LIN {X -0.164,Y -450.887,Z 1407.566,A 0.000,B 0.000,C 90.000,E1 281.951} C_DIS
LIN {X -0.109,Y -452.134,Z 1407.563,A 0.000,B 0.000,C 90.000,E1 281.422} C_DIS
LIN {X -0.046,Y -452.993,Z 1407.561,A 0.000,B 0.000,C 90.000,E1 280.894} C_DIS
LIN {X 0.023,Y -453.472,Z 1407.558,A 0.000,B 0.000,C 90.000,E1 280.366} C_DIS
LIN {X 0.016,Y -453.459,Z 1407.555,A 0.000,B 0.000,C 90.000,E1 279.849} C_DIS
LIN {X 0.091,Y -452.973,Z 1407.552,A 0.000,B 0.000,C 90.000,E1 279.321} C_DIS
LIN {X 0.091,Y -451.933,Z 1407.549,A 0.000,B 0.000,C 90.000,E1 278.803} C_DIS
LIN {X 0.156,Y -450.386,Z 1407.546,A 0.000,B 0.000,C 90.000,E1 278.276} C_DIS
LIN {X 0.149,Y -448.152,Z 1407.543,A 0.000,B 0.000,C 90.000,E1 277.757} C_DIS
LIN {X 0.128,Y -445.154,Z 1407.540,A 0.000,B 0.000,C 90.000,E1 277.239} C_DIS
LIN {X -0.082,Y -443.358,Z 1407.539,A 0.000,B 0.000,C 90.000,E1 277.004} C_DIS
LIN {X -0.126,Y -439.024,Z 1407.536,A 0.000,B 0.000,C 90.000,E1 276.486} C_DIS
LIN {X 0.042,Y -436.474,Z 1407.534,A 0.000,B 0.000,C 90.000,E1 276.201} C_DIS
LIN {X 0.046,Y -430.491,Z 1407.532,A 0.000,B 0.000,C 90.000,E1 275.682} C_DIS
LIN {X 0.146,Y -424.269,Z 1407.529,A 0.000,B 0.000,C 90.000,E1 275.220} C_DIS
LIN {X -0.212,Y -417.873,Z 1407.527,A 0.000,B 0.000,C 90.000,E1 274.878} C_DIS
LIN {X 0.190,Y -411.195,Z 1407.525,A 0.000,B 0.000,C 90.000,E1 274.473} C_DIS
LIN {X -0.124,Y -401.382,Z 1407.523,A 0.000,B 0.000,C 90.000,E1 274.073} C_DIS
LIN {X -0.064,Y -391.586,Z 1407.520,A 0.000,B 0.000,C 90.000,E1 273.669} C_DIS
LIN {X -0.077,Y -378.690,Z 1407.518,A 0.000,B 0.000,C 90.000,E1 273.212} C_DIS
LIN {X -0.178,Y -368.306,Z 1407.516,A 0.000,B 0.000,C 90.000,E1 272.922} C_DIS
LIN {X 0.035,Y -357.753,Z 1407.515,A 0.000,B 0.000,C 90.000,E1 272.636} C_DIS
LIN {X -0.170,Y -346.589,Z 1407.514,A 0.000,B 0.000,C 90.000,E1 272.465} C_DIS
LIN {X -0.105,Y -332.924,Z 1407.513,A 0.000,B 0.000,C 90.000,E1 272.293} C_DIS
LIN {X 0.118,Y -317.949,Z 1407.512,A 0.000,B 0.000,C 90.000,E1 272.178} C_DIS
LIN {X 0.057,Y -313.232,Z 1407.512,A 0.000,B 0.000,C 90.000,E1 272.178} C_DIS
LIN {X 0.014,Y -181.233,Z 1407.512,A 0.000,B 0.000,C 90.000,E1 272.178} C_DIS
LIN {X -0.010,Y -181.571,Z 1407.503,A 0.000,B 0.000,C 90.000,E1 270.458} C_DIS
LIN {X -0.090,Y -180.932,Z 1407.479,A 0.000,B 0.000,C 90.000,E1 266.274} C_DIS
LIN {X -0.032,Y -180.906,Z 1407.474,A 0.000,B 0.000,C 90.000,E1 265.412} C_DIS
LIN {X 0.041,Y -180.705,Z 1407.470,A 0.000,B 0.000,C 90.000,E1 264.546} C_DIS
LIN {X -0.056,Y -178.791,Z 1407.442,A 0.000,B 0.000,C 90.000,E1 259.511} C_DIS
LIN {X 0.020,Y -175.837,Z 1407.413,A 0.000,B 0.000,C 90.000,E1 254.393} C_DIS
LIN {X 0.021,Y -172.026,Z 1407.385,A 0.000,B 0.000,C 90.000,E1 249.263} C_DIS
LIN {X -0.003,Y -171.453,Z 1407.380,A 0.000,B 0.000,C 90.000,E1 248.411} C_DIS
LIN {X -0.023,Y -167.687,Z 1407.356,A 0.000,B 0.000,C 90.000,E1 244.101} C_DIS
LIN {X -0.009,Y -166.367,Z 1407.346,A 0.000,B 0.000,C 90.000,E1 242.359} C_DIS
LIN {X -0.017,Y -163.098,Z 1407.327,A 0.000,B 0.000,C 90.000,E1 238.869} C_DIS
LIN {X 0.034,Y -161.043,Z 1407.312,A 0.000,B 0.000,C 90.000,E1 236.215} C_DIS
LIN {X 0.018,Y -157.780,Z 1407.293,A 0.000,B 0.000,C 90.000,E1 232.683} C_DIS
LIN {X 0.080,Y -155.817,Z 1407.278,A 0.000,B 0.000,C 90.000,E1 229.989} C_DIS
LIN {X -0.081,Y -152.069,Z 1407.253,A 0.000,B 0.000,C 90.000,E1 225.567} C_DIS
LIN {X -0.062,Y -150.319,Z 1407.238,A 0.000,B 0.000,C 90.000,E1 222.852} C_DIS
LIN {X -0.040,Y -147.061,Z 1407.213,A 0.000,B 0.000,C 90.000,E1 218.302} C_DIS
LIN {X 0.067,Y -145.638,Z 1407.198,A 0.000,B 0.000,C 90.000,E1 215.518} C_DIS
LIN {X 0.065,Y -143.020,Z 1407.172,A 0.000,B 0.000,C 90.000,E1 210.924} C_DIS
LIN {X -0.004,Y -141.646,Z 1407.151,A 0.000,B 0.000,C 90.000,E1 207.257} C_DIS
LIN {X 0.046,Y -139.442,Z 1407.115,A 0.000,B 0.000,C 90.000,E1 200.737} C_DIS
LIN {X -0.032,Y -139.175,Z 1407.105,A 0.000,B 0.000,C 90.000,E1 198.906} C_DIS
LIN {X -0.004,Y -138.319,Z 1407.053,A 0.000,B 0.000,C 90.000,E1 189.557} C_DIS
LIN {X 0.006,Y -139.470,Z 1407.006,A 0.000,B 0.000,C 90.000,E1 181.146} C_DIS
LIN {X -0.054,Y -141.040,Z 1406.975,A 0.000,B 0.000,C 90.000,E1 175.584} C_DIS
LIN {X 0.041,Y -142.409,Z 1406.960,A 0.000,B 0.000,C 90.000,E1 172.761} C_DIS
LIN {X -0.038,Y -144.642,Z 1406.934,A 0.000,B 0.000,C 90.000,E1 168.173} C_DIS
LIN {X 0.022,Y -147.839,Z 1406.909,A 0.000,B 0.000,C 90.000,E1 163.559} C_DIS
LIN {X -0.034,Y -150.536,Z 1406.888,A 0.000,B 0.000,C 90.000,E1 159.934} C_DIS
LIN {X -0.016,Y -154.000,Z 1406.868,A 0.000,B 0.000,C 90.000,E1 156.305} C_DIS
LIN {X 0.045,Y -157.413,Z 1406.848,A 0.000,B 0.000,C 90.000,E1 152.692} C_DIS
LIN {X 0.067,Y -161.624,Z 1406.829,A 0.000,B 0.000,C 90.000,E1 149.125} C_DIS
LIN {X 0.086,Y -165.819,Z 1406.809,A 0.000,B 0.000,C 90.000,E1 145.595} C_DIS
LIN {X 0.079,Y -170.788,Z 1406.790,A 0.000,B 0.000,C 90.000,E1 142.110} C_DIS
LIN {X -0.004,Y -175.659,Z 1406.771,A 0.000,B 0.000,C 90.000,E1 138.690} C_DIS
LIN {X -0.007,Y -181.273,Z 1406.752,A 0.000,B 0.000,C 90.000,E1 135.283} C_DIS
LIN {X -0.007,Y -186.748,Z 1406.733,A 0.000,B 0.000,C 90.000,E1 131.919} C_DIS
LIN {X -0.056,Y -191.344,Z 1406.719,A 0.000,B 0.000,C 90.000,E1 129.439} C_DIS
LIN {X -0.010,Y -197.180,Z 1406.701,A 0.000,B 0.000,C 90.000,E1 126.137} C_DIS
LIN {X 0.015,Y -199.638,Z 1406.694,A 0.000,B 0.000,C 90.000,E1 124.898} C_DIS
LIN {X -0.011,Y -310.460,Z 1406.694,A 0.000,B 0.000,C 90.000,E1 124.898} C_DIS
LIN {X 0.052,Y -316.081,Z 1406.693,A 0.000,B 0.000,C 90.000,E1 124.692} C_DIS
LIN {X 0.117,Y -318.647,Z 1406.692,A 0.000,B 0.000,C 90.000,E1 124.485} C_DIS
LIN {X -0.078,Y -322.451,Z 1406.689,A 0.000,B 0.000,C 90.000,E1 124.072} C_DIS
LIN {X 0.211,Y -324.301,Z 1406.688,A 0.000,B 0.000,C 90.000,E1 123.706} C_DIS
LIN {X 0.047,Y -325.742,Z 1406.686,A 0.000,B 0.000,C 90.000,E1 123.420} C_DIS
LIN {X -0.157,Y -338.662,Z 1406.667,A 0.000,B 0.000,C 90.000,E1 120.001} C_DIS
LIN {X -0.002,Y -350.683,Z 1406.651,A 0.000,B 0.000,C 90.000,E1 117.206} C_DIS
LIN {X -0.134,Y -364.162,Z 1406.636,A 0.000,B 0.000,C 90.000,E1 114.515} C_DIS
LIN {X -0.121,Y -377.467,Z 1406.623,A 0.000,B 0.000,C 90.000,E1 112.153} C_DIS
LIN {X 0.091,Y -392.109,Z 1406.610,A 0.000,B 0.000,C 90.000,E1 109.812} C_DIS
LIN {X -0.098,Y -408.194,Z 1406.598,A 0.000,B 0.000,C 90.000,E1 107.583} C_DIS
LIN {X -0.012,Y -425.832,Z 1406.585,A 0.000,B 0.000,C 90.000,E1 105.371} C_DIS
LIN {X -0.082,Y -445.088,Z 1406.573,A 0.000,B 0.000,C 90.000,E1 103.244} C_DIS
LIN {X 0.011,Y -465.219,Z 1406.563,A 0.000,B 0.000,C 90.000,E1 101.243} C_DIS
LIN {X 0.182,Y -483.286,Z 1406.553,A 0.000,B 0.000,C 90.000,E1 99.613} C_DIS
LIN {X -0.157,Y -485.624,Z 1406.552,A 0.000,B 0.000,C 90.000,E1 99.434} C_DIS
LIN {X -0.097,Y -487.395,Z 1406.551,A 0.000,B 0.000,C 90.000,E1 99.208} C_DIS
LIN {X -0.205,Y -488.920,Z 1406.550,A 0.000,B 0.000,C 90.000,E1 98.973} C_DIS
LIN {X 0.096,Y -490.057,Z 1406.548,A 0.000,B 0.000,C 90.000,E1 98.690} C_DIS
LIN {X -0.102,Y -491.406,Z 1406.546,A 0.000,B 0.000,C 90.000,E1 98.219} C_DIS
LIN {X 0.121,Y -491.715,Z 1406.543,A 0.000,B 0.000,C 90.000,E1 97.701} C_DIS
LIN {X -0.136,Y -491.034,Z 1406.540,A 0.000,B 0.000,C 90.000,E1 97.239} C_DIS
LIN {X 0.097,Y -489.256,Z 1406.537,A 0.000,B 0.000,C 90.000,E1 96.720} C_DIS
LIN {X -0.004,Y -487.849,Z 1406.536,A 0.000,B 0.000,C 90.000,E1 96.486} C_DIS
LIN {X -0.036,Y -468.285,Z 1406.519,A 0.000,B 0.000,C 90.000,E1 93.498} C_DIS
LIN {X 0.108,Y -461.753,Z 1406.514,A 0.000,B 0.000,C 90.000,E1 92.465} C_DIS
LIN {X -0.208,Y -440.357,Z 1406.495,A 0.000,B 0.000,C 90.000,E1 89.141} C_DIS
LIN {X 0.076,Y -429.683,Z 1406.485,A 0.000,B 0.000,C 90.000,E1 87.249} C_DIS
LIN {X 0.154,Y -418.808,Z 1406.474,A 0.000,B 0.000,C 90.000,E1 85.355} C_DIS
LIN {X 0.081,Y -407.789,Z 1406.464,A 0.000,B 0.000,C 90.000,E1 83.451} C_DIS
LIN {X 0.192,Y -396.699,Z 1406.453,A 0.000,B 0.000,C 90.000,E1 81.489} C_DIS
LIN {X 0.132,Y -387.026,Z 1406.443,A 0.000,B 0.000,C 90.000,E1 79.803} C_DIS
LIN {X -0.003,Y -375.657,Z 1406.432,A 0.000,B 0.000,C 90.000,E1 77.813} C_DIS
LIN {X 0.077,Y -364.284,Z 1406.421,A 0.000,B 0.000,C 90.000,E1 75.755} C_DIS
LIN {X 0.049,Y -354.447,Z 1406.411,A 0.000,B 0.000,C 90.000,E1 73.976} C_DIS
LIN {X -0.058,Y -344.544,Z 1406.401,A 0.000,B 0.000,C 90.000,E1 72.181} C_DIS
LIN {X 0.078,Y -334.556,Z 1406.391,A 0.000,B 0.000,C 90.000,E1 70.315} C_DIS
LIN {X 0.057,Y -318.235,Z 1406.373,A 0.000,B 0.000,C 90.000,E1 67.177} C_DIS
LIN {X 0.021,Y -304.503,Z 1406.357,A 0.000,B 0.000,C 90.000,E1 64.280} C_DIS
LIN {X 0.023,Y -293.573,Z 1406.343,A 0.000,B 0.000,C 90.000,E1 61.641} C_DIS
LIN {X -0.024,Y -281.325,Z 1406.324,A 0.000,B 0.000,C 90.000,E1 58.280} C_DIS
LIN {X -0.014,Y -271.322,Z 1406.307,A 0.000,B 0.000,C 90.000,E1 55.182} C_DIS
LIN {X -0.104,Y -260.957,Z 1406.287,A 0.000,B 0.000,C 90.000,E1 51.698} C_DIS
LIN {X 0.091,Y -251.179,Z 1406.267,A 0.000,B 0.000,C 90.000,E1 48.081} C_DIS
LIN {X 0.115,Y -242.158,Z 1406.247,A 0.000,B 0.000,C 90.000,E1 44.433} C_DIS
LIN {X 0.036,Y -234.059,Z 1406.226,A 0.000,B 0.000,C 90.000,E1 40.744} C_DIS
LIN {X -0.040,Y -226.822,Z 1406.205,A 0.000,B 0.000,C 90.000,E1 36.996} C_DIS
LIN {X -0.010,Y -220.392,Z 1406.184,A 0.000,B 0.000,C 90.000,E1 33.166} C_DIS
LIN {X 0.026,Y -214.864,Z 1406.163,A 0.000,B 0.000,C 90.000,E1 29.283} C_DIS
LIN {X 0.135,Y -210.199,Z 1406.141,A 0.000,B 0.000,C 90.000,E1 25.335} C_DIS
LIN {X 0.044,Y -205.914,Z 1406.115,A 0.000,B 0.000,C 90.000,E1 20.610} C_DIS
LIN {X -0.045,Y -202.753,Z 1406.088,A 0.000,B 0.000,C 90.000,E1 15.843} C_DIS
LIN {X -0.046,Y -200.755,Z 1406.066,A 0.000,B 0.000,C 90.000,E1 11.827} C_DIS
LIN {X 0.077,Y -199.136,Z 1406.043,A 0.000,B 0.000,C 90.000,E1 7.757} C_DIS
LIN {X 0.020,Y -197.815,Z 1406.021,A 0.000,B 0.000,C 90.000,E1 3.726} C_DIS
LIN {X -0.036,Y -196.886,Z 1405.997,A 0.000,B 0.000,C 90.000,E1 359.542} C_DIS
LIN {X -0.050,Y -196.289,Z 1405.970,A 0.000,B 0.000,C 90.000,E1 354.666} C_DIS
LIN {X 0.067,Y -196.501,Z 1405.943,A 0.000,B 0.000,C 90.000,E1 349.746} C_DIS
LIN {X 0.116,Y -198.640,Z 1405.902,A 0.000,B 0.000,C 90.000,E1 342.417} C_DIS
LIN {X -0.055,Y -201.702,Z 1405.875,A 0.000,B 0.000,C 90.000,E1 337.614} C_DIS
LIN {X -0.023,Y -205.507,Z 1405.853,A 0.000,B 0.000,C 90.000,E1 333.589} C_DIS
LIN {X -0.055,Y -210.394,Z 1405.831,A 0.000,B 0.000,C 90.000,E1 329.616} C_DIS
LIN {X -0.040,Y -216.574,Z 1405.809,A 0.000,B 0.000,C 90.000,E1 325.674} C_DIS
LIN {X -0.019,Y -222.598,Z 1405.792,A 0.000,B 0.000,C 90.000,E1 322.557} C_DIS
LIN {X 0.080,Y -229.516,Z 1405.775,A 0.000,B 0.000,C 90.000,E1 319.461} C_DIS
LIN {X 0.117,Y -238.333,Z 1405.756,A 0.000,B 0.000,C 90.000,E1 316.053} C_DIS
LIN {X -0.096,Y -248.303,Z 1405.738,A 0.000,B 0.000,C 90.000,E1 312.771} C_DIS
LIN {X -0.027,Y -258.345,Z 1405.721,A 0.000,B 0.000,C 90.000,E1 309.850} C_DIS
LIN {X -0.088,Y -270.900,Z 1405.704,A 0.000,B 0.000,C 90.000,E1 306.664} C_DIS
LIN {X 0.116,Y -280.302,Z 1405.692,A 0.000,B 0.000,C 90.000,E1 304.532} C_DIS
LIN {X 0.091,Y -287.165,Z 1405.684,A 0.000,B 0.000,C 90.000,E1 303.166} C_DIS
LIN {X 0.144,Y -296.748,Z 1405.675,A 0.000,B 0.000,C 90.000,E1 301.465} C_DIS
LIN {X 0.175,Y -305.354,Z 1405.668,A 0.000,B 0.000,C 90.000,E1 300.129} C_DIS
LIN {X -0.112,Y -314.850,Z 1405.660,A 0.000,B 0.000,C 90.000,E1 298.871} C_DIS
LIN {X -0.129,Y -325.425,Z 1405.653,A 0.000,B 0.000,C 90.000,E1 297.590} C_DIS
LIN {X -0.149,Y -347.264,Z 1405.640,A 0.000,B 0.000,C 90.000,E1 295.207} C_DIS
LIN {X -0.068,Y -360.771,Z 1405.632,A 0.000,B 0.000,C 90.000,E1 293.770} C_DIS
LIN {X -0.063,Y -371.276,Z 1405.626,A 0.000,B 0.000,C 90.000,E1 292.642} C_DIS
LIN {X 0.059,Y -381.612,Z 1405.619,A 0.000,B 0.000,C 90.000,E1 291.482} C_DIS
LIN {X -0.077,Y -394.201,Z 1405.611,A 0.000,B 0.000,C 90.000,E1 290.066} C_DIS
LIN {X 0.079,Y -414.125,Z 1405.599,A 0.000,B 0.000,C 90.000,E1 287.819} C_DIS
LIN {X 0.165,Y -421.495,Z 1405.594,A 0.000,B 0.000,C 90.000,E1 286.985} C_DIS
LIN {X -0.032,Y -428.273,Z 1405.590,A 0.000,B 0.000,C 90.000,E1 286.205} C_DIS
LIN {X -0.001,Y -432.410,Z 1405.587,A 0.000,B 0.000,C 90.000,E1 285.662} C_DIS
LIN {X -0.063,Y -436.154,Z 1405.584,A 0.000,B 0.000,C 90.000,E1 285.134} C_DIS
LIN {X 0.219,Y -441.051,Z 1405.580,A 0.000,B 0.000,C 90.000,E1 284.300} C_DIS
LIN {X -0.215,Y -443.860,Z 1405.577,A 0.000,B 0.000,C 90.000,E1 283.828} C_DIS
LIN {X 0.027,Y -447.401,Z 1405.572,A 0.000,B 0.000,C 90.000,E1 283.008} C_DIS
LIN {X 0.067,Y -449.377,Z 1405.569,A 0.000,B 0.000,C 90.000,E1 282.479} C_DIS
LIN {X 0.112,Y -450.991,Z 1405.567,A 0.000,B 0.000,C 90.000,E1 281.951} C_DIS
LIN {X 0.169,Y -452.230,Z 1405.564,A 0.000,B 0.000,C 90.000,E1 281.422} C_DIS
LIN {X -0.212,Y -453.131,Z 1405.561,A 0.000,B 0.000,C 90.000,E1 280.950} C_DIS
LIN {X -0.142,Y -453.645,Z 1405.558,A 0.000,B 0.000,C 90.000,E1 280.423} C_DIS
LIN {X -0.150,Y -453.657,Z 1405.555,A 0.000,B 0.000,C 90.000,E1 279.905} C_DIS
LIN {X -0.075,Y -453.234,Z 1405.552,A 0.000,B 0.000,C 90.000,E1 279.378} C_DIS
LIN {X -0.074,Y -452.292,Z 1405.549,A 0.000,B 0.000,C 90.000,E1 278.859} C_DIS
LIN {X -0.071,Y -450.785,Z 1405.546,A 0.000,B 0.000,C 90.000,E1 278.341} C_DIS
LIN {X -0.012,Y -448.649,Z 1405.543,A 0.000,B 0.000,C 90.000,E1 277.814} C_DIS
LIN {X -0.024,Y -445.765,Z 1405.541,A 0.000,B 0.000,C 90.000,E1 277.296} C_DIS
LIN {X -0.054,Y -442.041,Z 1405.538,A 0.000,B 0.000,C 90.000,E1 276.777} C_DIS
LIN {X -0.102,Y -437.324,Z 1405.535,A 0.000,B 0.000,C 90.000,E1 276.258} C_DIS
LIN {X 0.115,Y -434.562,Z 1405.533,A 0.000,B 0.000,C 90.000,E1 275.967} C_DIS
LIN {X -0.139,Y -428.517,Z 1405.531,A 0.000,B 0.000,C 90.000,E1 275.511} C_DIS
LIN {X 0.120,Y -422.247,Z 1405.528,A 0.000,B 0.000,C 90.000,E1 275.049} C_DIS
LIN {X -0.075,Y -415.762,Z 1405.526,A 0.000,B 0.000,C 90.000,E1 274.702} C_DIS
LIN {X 0.148,Y -405.811,Z 1405.523,A 0.000,B 0.000,C 90.000,E1 274.188} C_DIS
LIN {X 0.094,Y -396.109,Z 1405.521,A 0.000,B 0.000,C 90.000,E1 273.784} C_DIS
LIN {X -0.108,Y -386.263,Z 1405.519,A 0.000,B 0.000,C 90.000,E1 273.440} C_DIS
LIN {X -0.010,Y -376.360,Z 1405.517,A 0.000,B 0.000,C 90.000,E1 273.094} C_DIS
LIN {X 0.172,Y -369.429,Z 1405.516,A 0.000,B 0.000,C 90.000,E1 272.865} C_DIS
LIN {X 0.019,Y -358.758,Z 1405.515,A 0.000,B 0.000,C 90.000,E1 272.636} C_DIS
LIN {X 0.165,Y -347.772,Z 1405.514,A 0.000,B 0.000,C 90.000,E1 272.407} C_DIS
LIN {X -0.119,Y -334.120,Z 1405.513,A 0.000,B 0.000,C 90.000,E1 272.293} C_DIS
LIN {X 0.108,Y -321.060,Z 1405.512,A 0.000,B 0.000,C 90.000,E1 272.178} C_DIS
LIN {X 0.010,Y -313.166,Z 1405.512,A 0.000,B 0.000,C 90.000,E1 272.178} C_DIS
LIN {X -0.016,Y -181.234,Z 1405.512,A 0.000,B 0.000,C 90.000,E1 272.178} C_DIS
LIN {X -0.034,Y -181.572,Z 1405.502,A 0.000,B 0.000,C 90.000,E1 270.458} C_DIS
LIN {X -0.056,Y -180.906,Z 1405.474,A 0.000,B 0.000,C 90.000,E1 265.412} C_DIS
LIN {X 0.018,Y -180.701,Z 1405.470,A 0.000,B 0.000,C 90.000,E1 264.546} C_DIS
LIN {X -0.081,Y -178.786,Z 1405.442,A 0.000,B 0.000,C 90.000,E1 259.511} C_DIS
LIN {X -0.003,Y -175.833,Z 1405.413,A 0.000,B 0.000,C 90.000,E1 254.393} C_DIS
LIN {X -0.002,Y -172.022,Z 1405.385,A 0.000,B 0.000,C 90.000,E1 249.263} C_DIS
LIN {X -0.026,Y -171.447,Z 1405.380,A 0.000,B 0.000,C 90.000,E1 248.411} C_DIS
LIN {X 0.028,Y -167.681,Z 1405.356,A 0.000,B 0.000,C 90.000,E1 244.076} C_DIS
LIN {X -0.032,Y -166.358,Z 1405.346,A 0.000,B 0.000,C 90.000,E1 242.359} C_DIS
LIN {X -0.039,Y -163.091,Z 1405.327,A 0.000,B 0.000,C 90.000,E1 238.869} C_DIS
LIN {X 0.012,Y -161.035,Z 1405.312,A 0.000,B 0.000,C 90.000,E1 236.215} C_DIS
LIN {X -0.005,Y -157.774,Z 1405.293,A 0.000,B 0.000,C 90.000,E1 232.683} C_DIS
LIN {X 0.058,Y -155.812,Z 1405.278,A 0.000,B 0.000,C 90.000,E1 229.989} C_DIS
LIN {X 0.006,Y -152.063,Z 1405.253,A 0.000,B 0.000,C 90.000,E1 225.526} C_DIS
LIN {X -0.083,Y -150.313,Z 1405.238,A 0.000,B 0.000,C 90.000,E1 222.852} C_DIS
LIN {X 0.054,Y -147.056,Z 1405.213,A 0.000,B 0.000,C 90.000,E1 218.257} C_DIS
LIN {X 0.046,Y -145.634,Z 1405.197,A 0.000,B 0.000,C 90.000,E1 215.518} C_DIS
LIN {X 0.045,Y -143.017,Z 1405.172,A 0.000,B 0.000,C 90.000,E1 210.924} C_DIS
LIN {X -0.025,Y -141.643,Z 1405.151,A 0.000,B 0.000,C 90.000,E1 207.257} C_DIS
LIN {X 0.026,Y -139.440,Z 1405.115,A 0.000,B 0.000,C 90.000,E1 200.737} C_DIS
LIN {X -0.052,Y -139.173,Z 1405.105,A 0.000,B 0.000,C 90.000,E1 198.906} C_DIS
LIN {X -0.024,Y -138.318,Z 1405.053,A 0.000,B 0.000,C 90.000,E1 189.557} C_DIS
LIN {X -0.015,Y -139.472,Z 1405.006,A 0.000,B 0.000,C 90.000,E1 181.146} C_DIS
LIN {X 0.066,Y -141.044,Z 1404.975,A 0.000,B 0.000,C 90.000,E1 175.527} C_DIS
LIN {X 0.021,Y -142.413,Z 1404.960,A 0.000,B 0.000,C 90.000,E1 172.761} C_DIS
LIN {X -0.059,Y -144.648,Z 1404.934,A 0.000,B 0.000,C 90.000,E1 168.173} C_DIS
LIN {X 0.001,Y -147.844,Z 1404.909,A 0.000,B 0.000,C 90.000,E1 163.559} C_DIS
LIN {X -0.056,Y -150.543,Z 1404.888,A 0.000,B 0.000,C 90.000,E1 159.934} C_DIS
LIN {X -0.037,Y -154.008,Z 1404.868,A 0.000,B 0.000,C 90.000,E1 156.305} C_DIS
LIN {X 0.022,Y -157.423,Z 1404.848,A 0.000,B 0.000,C 90.000,E1 152.692} C_DIS
LIN {X 0.045,Y -161.634,Z 1404.829,A 0.000,B 0.000,C 90.000,E1 149.125} C_DIS
LIN {X 0.063,Y -165.829,Z 1404.809,A 0.000,B 0.000,C 90.000,E1 145.595} C_DIS
LIN {X 0.055,Y -170.800,Z 1404.790,A 0.000,B 0.000,C 90.000,E1 142.110} C_DIS
LIN {X -0.027,Y -175.670,Z 1404.771,A 0.000,B 0.000,C 90.000,E1 138.690} C_DIS
LIN {X 0.097,Y -181.284,Z 1404.751,A 0.000,B 0.000,C 90.000,E1 135.243} C_DIS
LIN {X -0.031,Y -186.762,Z 1404.733,A 0.000,B 0.000,C 90.000,E1 131.919} C_DIS
LIN {X 0.041,Y -191.356,Z 1404.719,A 0.000,B 0.000,C 90.000,E1 129.402} C_DIS
LIN {X -0.035,Y -197.194,Z 1404.701,A 0.000,B 0.000,C 90.000,E1 126.137} C_DIS
LIN {X 0.077,Y -199.601,Z 1404.694,A 0.000,B 0.000,C 90.000,E1 124.898} C_DIS
LIN {X 0.087,Y -310.119,Z 1404.694,A 0.000,B 0.000,C 90.000,E1 124.898} C_DIS
LIN {X -0.048,Y -311.871,Z 1404.694,A 0.000,B 0.000,C 90.000,E1 124.898} C_DIS
LIN {X 0.013,Y -316.366,Z 1404.693,A 0.000,B 0.000,C 90.000,E1 124.692} C_DIS
LIN {X 0.077,Y -318.822,Z 1404.692,A 0.000,B 0.000,C 90.000,E1 124.485} C_DIS
LIN {X -0.034,Y -322.641,Z 1404.689,A 0.000,B 0.000,C 90.000,E1 124.040} C_DIS
LIN {X 0.042,Y -324.457,Z 1404.687,A 0.000,B 0.000,C 90.000,E1 123.706} C_DIS
LIN {X 0.121,Y -325.868,Z 1404.686,A 0.000,B 0.000,C 90.000,E1 123.372} C_DIS
LIN {X -0.035,Y -337.529,Z 1404.668,A 0.000,B 0.000,C 90.000,E1 120.256} C_DIS
LIN {X 0.090,Y -349.408,Z 1404.653,A 0.000,B 0.000,C 90.000,E1 117.462} C_DIS
LIN {X -0.078,Y -362.742,Z 1404.638,A 0.000,B 0.000,C 90.000,E1 114.771} C_DIS
LIN {X 0.047,Y -375.903,Z 1404.624,A 0.000,B 0.000,C 90.000,E1 112.386} C_DIS
LIN {X 0.083,Y -390.393,Z 1404.612,A 0.000,B 0.000,C 90.000,E1 110.066} C_DIS
LIN {X -0.017,Y -406.312,Z 1404.599,A 0.000,B 0.000,C 90.000,E1 107.819} C_DIS
LIN {X 0.023,Y -423.773,Z 1404.587,A 0.000,B 0.000,C 90.000,E1 105.607} C_DIS
LIN {X -0.026,Y -442.876,Z 1404.575,A 0.000,B 0.000,C 90.000,E1 103.467} C_DIS
LIN {X -0.190,Y -462.943,Z 1404.564,A 0.000,B 0.000,C 90.000,E1 101.478} C_DIS
LIN {X -0.029,Y -483.550,Z 1404.553,A 0.000,B 0.000,C 90.000,E1 99.613} C_DIS
LIN {X 0.112,Y -485.789,Z 1404.552,A 0.000,B 0.000,C 90.000,E1 99.378} C_DIS
LIN {X 0.175,Y -487.486,Z 1404.551,A 0.000,B 0.000,C 90.000,E1 99.151} C_DIS
LIN {X 0.069,Y -488.951,Z 1404.550,A 0.000,B 0.000,C 90.000,E1 98.916} C_DIS
LIN {X -0.038,Y -490.040,Z 1404.548,A 0.000,B 0.000,C 90.000,E1 98.681} C_DIS
LIN {X 0.176,Y -491.312,Z 1404.545,A 0.000,B 0.000,C 90.000,E1 98.163} C_DIS
LIN {X -0.090,Y -491.553,Z 1404.543,A 0.000,B 0.000,C 90.000,E1 97.701} C_DIS
LIN {X 0.141,Y -490.804,Z 1404.540,A 0.000,B 0.000,C 90.000,E1 97.182} C_DIS
LIN {X -0.113,Y -488.940,Z 1404.537,A 0.000,B 0.000,C 90.000,E1 96.720} C_DIS
LIN {X -0.214,Y -487.476,Z 1404.536,A 0.000,B 0.000,C 90.000,E1 96.486} C_DIS
LIN {X 0.217,Y -467.918,Z 1404.519,A 0.000,B 0.000,C 90.000,E1 93.440} C_DIS
LIN {X 0.145,Y -459.666,Z 1404.512,A 0.000,B 0.000,C 90.000,E1 92.178} C_DIS
LIN {X 0.012,Y -439.998,Z 1404.495,A 0.000,B 0.000,C 90.000,E1 89.083} C_DIS
LIN {X -0.146,Y -429.339,Z 1404.485,A 0.000,B 0.000,C 90.000,E1 87.249} C_DIS
LIN {X -0.068,Y -418.503,Z 1404.474,A 0.000,B 0.000,C 90.000,E1 85.355} C_DIS
LIN {X -0.142,Y -407.532,Z 1404.464,A 0.000,B 0.000,C 90.000,E1 83.451} C_DIS
LIN {X -0.030,Y -396.456,Z 1404.453,A 0.000,B 0.000,C 90.000,E1 81.489} C_DIS
LIN {X -0.088,Y -386.792,Z 1404.443,A 0.000,B 0.000,C 90.000,E1 79.803} C_DIS
LIN {X 0.145,Y -375.453,Z 1404.432,A 0.000,B 0.000,C 90.000,E1 77.757} C_DIS
LIN {X -0.139,Y -364.079,Z 1404.421,A 0.000,B 0.000,C 90.000,E1 75.755} C_DIS
LIN {X -0.165,Y -354.215,Z 1404.411,A 0.000,B 0.000,C 90.000,E1 73.976} C_DIS
LIN {X 0.057,Y -344.308,Z 1404.401,A 0.000,B 0.000,C 90.000,E1 72.127} C_DIS
LIN {X -0.019,Y -334.294,Z 1404.391,A 0.000,B 0.000,C 90.000,E1 70.296} C_DIS
LIN {X -0.151,Y -317.969,Z 1404.373,A 0.000,B 0.000,C 90.000,E1 67.177} C_DIS
LIN {X 0.121,Y -302.841,Z 1404.355,A 0.000,B 0.000,C 90.000,E1 63.896} C_DIS
LIN {X 0.080,Y -292.078,Z 1404.340,A 0.000,B 0.000,C 90.000,E1 61.257} C_DIS
LIN {X 0.126,Y -280.013,Z 1404.322,A 0.000,B 0.000,C 90.000,E1 57.867} C_DIS
LIN {X 0.011,Y -271.202,Z 1404.306,A 0.000,B 0.000,C 90.000,E1 55.135} C_DIS
LIN {X 0.069,Y -260.886,Z 1404.287,A 0.000,B 0.000,C 90.000,E1 51.618} C_DIS
LIN {X -0.097,Y -251.135,Z 1404.267,A 0.000,B 0.000,C 90.000,E1 48.081} C_DIS
LIN {X -0.068,Y -242.146,Z 1404.247,A 0.000,B 0.000,C 90.000,E1 44.433} C_DIS
LIN {X 0.037,Y -234.077,Z 1404.226,A 0.000,B 0.000,C 90.000,E1 40.701} C_DIS
LIN {X -0.030,Y -226.866,Z 1404.205,A 0.000,B 0.000,C 90.000,E1 36.950} C_DIS
LIN {X 0.131,Y -220.480,Z 1404.184,A 0.000,B 0.000,C 90.000,E1 33.086} C_DIS
LIN {X -0.026,Y -214.981,Z 1404.162,A 0.000,B 0.000,C 90.000,E1 29.255} C_DIS
LIN {X -0.015,Y -210.377,Z 1404.141,A 0.000,B 0.000,C 90.000,E1 25.335} C_DIS
LIN {X -0.096,Y -206.140,Z 1404.114,A 0.000,B 0.000,C 90.000,E1 20.610} C_DIS
LIN {X 0.022,Y -203.037,Z 1404.088,A 0.000,B 0.000,C 90.000,E1 15.788} C_DIS
LIN {X 0.032,Y -201.072,Z 1404.065,A 0.000,B 0.000,C 90.000,E1 11.771} C_DIS
LIN {X -0.030,Y -199.452,Z 1404.043,A 0.000,B 0.000,C 90.000,E1 7.757} C_DIS
LIN {X -0.078,Y -198.140,Z 1404.021,A 0.000,B 0.000,C 90.000,E1 3.726} C_DIS
LIN {X -0.036,Y -197.190,Z 1403.997,A 0.000,B 0.000,C 90.000,E1 359.542} C_DIS
LIN {X -0.040,Y -196.550,Z 1403.970,A 0.000,B 0.000,C 90.000,E1 354.666} C_DIS
LIN {X 0.087,Y -196.734,Z 1403.943,A 0.000,B 0.000,C 90.000,E1 349.746} C_DIS
LIN {X -0.100,Y -198.883,Z 1403.903,A 0.000,B 0.000,C 90.000,E1 342.489} C_DIS
LIN {X -0.012,Y -201.927,Z 1403.876,A 0.000,B 0.000,C 90.000,E1 337.614} C_DIS
LIN {X 0.027,Y -205.729,Z 1403.853,A 0.000,B 0.000,C 90.000,E1 333.589} C_DIS
LIN {X 0.005,Y -210.613,Z 1403.831,A 0.000,B 0.000,C 90.000,E1 329.616} C_DIS
LIN {X 0.028,Y -216.789,Z 1403.809,A 0.000,B 0.000,C 90.000,E1 325.674} C_DIS
LIN {X 0.035,Y -221.194,Z 1403.796,A 0.000,B 0.000,C 90.000,E1 323.336} C_DIS
LIN {X -0.040,Y -227.890,Z 1403.779,A 0.000,B 0.000,C 90.000,E1 320.275} C_DIS
LIN {X -0.047,Y -236.448,Z 1403.760,A 0.000,B 0.000,C 90.000,E1 316.863} C_DIS
LIN {X 0.021,Y -246.105,Z 1403.742,A 0.000,B 0.000,C 90.000,E1 313.500} C_DIS
LIN {X -0.150,Y -255.833,Z 1403.725,A 0.000,B 0.000,C 90.000,E1 310.620} C_DIS
LIN {X 0.045,Y -268.089,Z 1403.708,A 0.000,B 0.000,C 90.000,E1 307.363} C_DIS
LIN {X 0.034,Y -277.137,Z 1403.696,A 0.000,B 0.000,C 90.000,E1 305.264} C_DIS
LIN {X -0.153,Y -285.453,Z 1403.686,A 0.000,B 0.000,C 90.000,E1 303.579} C_DIS
LIN {X -0.129,Y -294.774,Z 1403.677,A 0.000,B 0.000,C 90.000,E1 301.878} C_DIS
LIN {X -0.130,Y -303.168,Z 1403.670,A 0.000,B 0.000,C 90.000,E1 300.541} C_DIS
LIN {X -0.022,Y -312.381,Z 1403.662,A 0.000,B 0.000,C 90.000,E1 299.205} C_DIS
LIN {X -0.059,Y -319.685,Z 1403.657,A 0.000,B 0.000,C 90.000,E1 298.281} C_DIS
LIN {X 0.030,Y -344.032,Z 1403.642,A 0.000,B 0.000,C 90.000,E1 295.540} C_DIS
LIN {X -0.110,Y -357.565,Z 1403.634,A 0.000,B 0.000,C 90.000,E1 294.131} C_DIS
LIN {X -0.102,Y -368.124,Z 1403.628,A 0.000,B 0.000,C 90.000,E1 293.003} C_DIS
LIN {X 0.031,Y -378.528,Z 1403.621,A 0.000,B 0.000,C 90.000,E1 291.844} C_DIS
LIN {X -0.088,Y -391.142,Z 1403.613,A 0.000,B 0.000,C 90.000,E1 290.429} C_DIS
LIN {X 0.203,Y -408.577,Z 1403.602,A 0.000,B 0.000,C 90.000,E1 288.417} C_DIS
LIN {X -0.207,Y -418.361,Z 1403.597,A 0.000,B 0.000,C 90.000,E1 287.402} C_DIS
LIN {X 0.028,Y -425.472,Z 1403.592,A 0.000,B 0.000,C 90.000,E1 286.551} C_DIS
LIN {X 0.082,Y -431.912,Z 1403.588,A 0.000,B 0.000,C 90.000,E1 285.733} C_DIS
LIN {X -0.095,Y -437.493,Z 1403.583,A 0.000,B 0.000,C 90.000,E1 284.954} C_DIS
LIN {X 0.192,Y -442.247,Z 1403.579,A 0.000,B 0.000,C 90.000,E1 284.120} C_DIS
LIN {X -0.010,Y -446.124,Z 1403.574,A 0.000,B 0.000,C 90.000,E1 283.355} C_DIS
LIN {X -0.183,Y -449.278,Z 1403.570,A 0.000,B 0.000,C 90.000,E1 282.591} C_DIS
LIN {X -0.141,Y -450.930,Z 1403.567,A 0.000,B 0.000,C 90.000,E1 282.063} C_DIS
LIN {X -0.087,Y -452.258,Z 1403.564,A 0.000,B 0.000,C 90.000,E1 281.535} C_DIS
LIN {X -0.025,Y -453.220,Z 1403.561,A 0.000,B 0.000,C 90.000,E1 281.007} C_DIS
LIN {X -0.039,Y -453.764,Z 1403.558,A 0.000,B 0.000,C 90.000,E1 280.489} C_DIS
LIN {X 0.037,Y -453.894,Z 1403.555,A 0.000,B 0.000,C 90.000,E1 279.962} C_DIS
LIN {X 0.037,Y -453.553,Z 1403.552,A 0.000,B 0.000,C 90.000,E1 279.443} C_DIS
LIN {X 0.112,Y -452.710,Z 1403.550,A 0.000,B 0.000,C 90.000,E1 278.916} C_DIS
LIN {X 0.115,Y -451.321,Z 1403.547,A 0.000,B 0.000,C 90.000,E1 278.398} C_DIS
LIN {X 0.177,Y -449.329,Z 1403.544,A 0.000,B 0.000,C 90.000,E1 277.871} C_DIS
LIN {X 0.166,Y -446.626,Z 1403.541,A 0.000,B 0.000,C 90.000,E1 277.352} C_DIS
LIN {X 0.138,Y -443.121,Z 1403.538,A 0.000,B 0.000,C 90.000,E1 276.834} C_DIS
LIN {X 0.093,Y -438.611,Z 1403.535,A 0.000,B 0.000,C 90.000,E1 276.315} C_DIS
LIN {X 0.026,Y -432.959,Z 1403.532,A 0.000,B 0.000,C 90.000,E1 275.796} C_DIS
LIN {X -0.053,Y -426.827,Z 1403.530,A 0.000,B 0.000,C 90.000,E1 275.334} C_DIS
LIN {X -0.131,Y -420.541,Z 1403.527,A 0.000,B 0.000,C 90.000,E1 274.935} C_DIS
LIN {X 0.159,Y -413.930,Z 1403.525,A 0.000,B 0.000,C 90.000,E1 274.531} C_DIS
LIN {X 0.153,Y -404.144,Z 1403.523,A 0.000,B 0.000,C 90.000,E1 274.073} C_DIS
LIN {X 0.139,Y -394.357,Z 1403.521,A 0.000,B 0.000,C 90.000,E1 273.669} C_DIS
LIN {X 0.042,Y -384.746,Z 1403.519,A 0.000,B 0.000,C 90.000,E1 273.326} C_DIS
LIN {X 0.185,Y -374.728,Z 1403.517,A 0.000,B 0.000,C 90.000,E1 272.980} C_DIS
LIN {X -0.098,Y -364.219,Z 1403.515,A 0.000,B 0.000,C 90.000,E1 272.751} C_DIS
LIN {X -0.085,Y -353.429,Z 1403.514,A 0.000,B 0.000,C 90.000,E1 272.522} C_DIS
LIN {X -0.102,Y -341.482,Z 1403.513,A 0.000,B 0.000,C 90.000,E1 272.350} C_DIS
LIN {X -0.107,Y -328.345,Z 1403.512,A 0.000,B 0.000,C 90.000,E1 272.236} C_DIS
LIN {X -0.044,Y -312.540,Z 1403.512,A 0.000,B 0.000,C 90.000,E1 272.178} C_DIS
LIN {X -0.051,Y -181.236,Z 1403.512,A 0.000,B 0.000,C 90.000,E1 272.178} C_DIS
LIN {X -0.044,Y -181.571,Z 1403.502,A 0.000,B 0.000,C 90.000,E1 270.458} C_DIS
LIN {X -0.066,Y -180.906,Z 1403.474,A 0.000,B 0.000,C 90.000,E1 265.412} C_DIS
LIN {X 0.008,Y -180.700,Z 1403.470,A 0.000,B 0.000,C 90.000,E1 264.546} C_DIS
LIN {X 0.086,Y -178.785,Z 1403.442,A 0.000,B 0.000,C 90.000,E1 259.454} C_DIS
LIN {X -0.012,Y -175.831,Z 1403.413,A 0.000,B 0.000,C 90.000,E1 254.393} C_DIS
LIN {X -0.012,Y -172.020,Z 1403.385,A 0.000,B 0.000,C 90.000,E1 249.263} C_DIS
LIN {X -0.035,Y -171.444,Z 1403.380,A 0.000,B 0.000,C 90.000,E1 248.411} C_DIS
LIN {X 0.019,Y -167.679,Z 1403.356,A 0.000,B 0.000,C 90.000,E1 244.076} C_DIS
LIN {X -0.041,Y -166.355,Z 1403.346,A 0.000,B 0.000,C 90.000,E1 242.359} C_DIS
LIN {X -0.048,Y -163.088,Z 1403.327,A 0.000,B 0.000,C 90.000,E1 238.869} C_DIS
LIN {X 0.003,Y -161.032,Z 1403.312,A 0.000,B 0.000,C 90.000,E1 236.215} C_DIS
LIN {X -0.014,Y -157.771,Z 1403.293,A 0.000,B 0.000,C 90.000,E1 232.683} C_DIS
LIN {X 0.049,Y -155.809,Z 1403.278,A 0.000,B 0.000,C 90.000,E1 229.989} C_DIS
LIN {X -0.003,Y -152.061,Z 1403.253,A 0.000,B 0.000,C 90.000,E1 225.526} C_DIS
LIN {X 0.010,Y -150.310,Z 1403.238,A 0.000,B 0.000,C 90.000,E1 222.813} C_DIS
LIN {X 0.045,Y -147.054,Z 1403.213,A 0.000,B 0.000,C 90.000,E1 218.257} C_DIS
LIN {X 0.038,Y -145.632,Z 1403.197,A 0.000,B 0.000,C 90.000,E1 215.518} C_DIS
LIN {X 0.035,Y -143.015,Z 1403.172,A 0.000,B 0.000,C 90.000,E1 210.924} C_DIS
LIN {X -0.033,Y -141.642,Z 1403.151,A 0.000,B 0.000,C 90.000,E1 207.257} C_DIS
LIN {X 0.017,Y -139.440,Z 1403.115,A 0.000,B 0.000,C 90.000,E1 200.737} C_DIS
LIN {X -0.061,Y -139.173,Z 1403.105,A 0.000,B 0.000,C 90.000,E1 198.906} C_DIS
LIN {X -0.032,Y -138.318,Z 1403.053,A 0.000,B 0.000,C 90.000,E1 189.557} C_DIS
LIN {X -0.023,Y -139.471,Z 1403.006,A 0.000,B 0.000,C 90.000,E1 181.146} C_DIS
LIN {X 0.058,Y -141.045,Z 1402.975,A 0.000,B 0.000,C 90.000,E1 175.527} C_DIS
LIN {X 0.012,Y -142.416,Z 1402.960,A 0.000,B 0.000,C 90.000,E1 172.761} C_DIS
LIN {X -0.068,Y -144.650,Z 1402.934,A 0.000,B 0.000,C 90.000,E1 168.173} C_DIS
LIN {X -0.008,Y -147.846,Z 1402.909,A 0.000,B 0.000,C 90.000,E1 163.559} C_DIS
LIN {X 0.077,Y -150.545,Z 1402.888,A 0.000,B 0.000,C 90.000,E1 159.880} C_DIS
LIN {X -0.046,Y -154.011,Z 1402.868,A 0.000,B 0.000,C 90.000,E1 156.305} C_DIS
LIN {X 0.014,Y -157.426,Z 1402.848,A 0.000,B 0.000,C 90.000,E1 152.692} C_DIS
LIN {X 0.035,Y -161.638,Z 1402.828,A 0.000,B 0.000,C 90.000,E1 149.125} C_DIS
LIN {X 0.053,Y -165.833,Z 1402.809,A 0.000,B 0.000,C 90.000,E1 145.595} C_DIS
LIN {X 0.045,Y -170.805,Z 1402.790,A 0.000,B 0.000,C 90.000,E1 142.110} C_DIS
LIN {X -0.037,Y -175.676,Z 1402.770,A 0.000,B 0.000,C 90.000,E1 138.690} C_DIS
LIN {X 0.086,Y -181.289,Z 1402.751,A 0.000,B 0.000,C 90.000,E1 135.243} C_DIS
LIN {X -0.041,Y -186.767,Z 1402.733,A 0.000,B 0.000,C 90.000,E1 131.919} C_DIS
LIN {X 0.030,Y -191.362,Z 1402.719,A 0.000,B 0.000,C 90.000,E1 129.402} C_DIS
LIN {X -0.046,Y -197.200,Z 1402.701,A 0.000,B 0.000,C 90.000,E1 126.137} C_DIS
LIN {X -0.031,Y -199.569,Z 1402.694,A 0.000,B 0.000,C 90.000,E1 124.945} C_DIS
LIN {X -0.083,Y -310.080,Z 1402.694,A 0.000,B 0.000,C 90.000,E1 124.945} C_DIS
LIN {X -0.064,Y -312.532,Z 1402.694,A 0.000,B 0.000,C 90.000,E1 124.898} C_DIS
LIN {X -0.003,Y -316.572,Z 1402.693,A 0.000,B 0.000,C 90.000,E1 124.692} C_DIS
LIN {X 0.060,Y -318.947,Z 1402.692,A 0.000,B 0.000,C 90.000,E1 124.485} C_DIS
LIN {X 0.140,Y -322.773,Z 1402.689,A 0.000,B 0.000,C 90.000,E1 123.992} C_DIS
LIN {X -0.051,Y -324.540,Z 1402.687,A 0.000,B 0.000,C 90.000,E1 123.706} C_DIS
LIN {X 0.027,Y -325.916,Z 1402.685,A 0.000,B 0.000,C 90.000,E1 123.372} C_DIS
LIN {X -0.131,Y -337.573,Z 1402.668,A 0.000,B 0.000,C 90.000,E1 120.256} C_DIS
LIN {X -0.008,Y -349.459,Z 1402.653,A 0.000,B 0.000,C 90.000,E1 117.462} C_DIS
LIN {X -0.177,Y -362.801,Z 1402.637,A 0.000,B 0.000,C 90.000,E1 114.771} C_DIS
LIN {X -0.055,Y -375.971,Z 1402.624,A 0.000,B 0.000,C 90.000,E1 112.386} C_DIS
LIN {X -0.021,Y -390.469,Z 1402.611,A 0.000,B 0.000,C 90.000,E1 110.066} C_DIS
LIN {X -0.123,Y -406.398,Z 1402.599,A 0.000,B 0.000,C 90.000,E1 107.819} C_DIS
LIN {X -0.086,Y -423.869,Z 1402.587,A 0.000,B 0.000,C 90.000,E1 105.607} C_DIS
LIN {X -0.136,Y -442.981,Z 1402.575,A 0.000,B 0.000,C 90.000,E1 103.467} C_DIS
LIN {X 0.158,Y -463.052,Z 1402.564,A 0.000,B 0.000,C 90.000,E1 101.422} C_DIS
LIN {X -0.132,Y -483.662,Z 1402.553,A 0.000,B 0.000,C 90.000,E1 99.613} C_DIS
LIN {X -0.017,Y -485.859,Z 1402.552,A 0.000,B 0.000,C 90.000,E1 99.378} C_DIS
LIN {X 0.020,Y -487.525,Z 1402.551,A 0.000,B 0.000,C 90.000,E1 99.151} C_DIS
LIN {X -0.086,Y -488.942,Z 1402.549,A 0.000,B 0.000,C 90.000,E1 98.916} C_DIS
LIN {X -0.193,Y -489.993,Z 1402.548,A 0.000,B 0.000,C 90.000,E1 98.681} C_DIS
LIN {X 0.019,Y -491.204,Z 1402.545,A 0.000,B 0.000,C 90.000,E1 98.163} C_DIS
LIN {X -0.245,Y -491.390,Z 1402.543,A 0.000,B 0.000,C 90.000,E1 97.701} C_DIS
LIN {X -0.015,Y -490.584,Z 1402.540,A 0.000,B 0.000,C 90.000,E1 97.182} C_DIS
LIN {X 0.216,Y -488.649,Z 1402.537,A 0.000,B 0.000,C 90.000,E1 96.663} C_DIS
LIN {X -0.042,Y -485.428,Z 1402.534,A 0.000,B 0.000,C 90.000,E1 96.201} C_DIS
LIN {X 0.056,Y -467.575,Z 1402.519,A 0.000,B 0.000,C 90.000,E1 93.440} C_DIS
LIN {X -0.019,Y -459.301,Z 1402.512,A 0.000,B 0.000,C 90.000,E1 92.178} C_DIS
LIN {X 0.099,Y -441.230,Z 1402.496,A 0.000,B 0.000,C 90.000,E1 89.312} C_DIS
LIN {X 0.112,Y -429.048,Z 1402.484,A 0.000,B 0.000,C 90.000,E1 87.192} C_DIS
LIN {X 0.176,Y -418.247,Z 1402.474,A 0.000,B 0.000,C 90.000,E1 85.298} C_DIS
LIN {X 0.091,Y -407.304,Z 1402.463,A 0.000,B 0.000,C 90.000,E1 83.394} C_DIS
LIN {X 0.189,Y -396.253,Z 1402.453,A 0.000,B 0.000,C 90.000,E1 81.432} C_DIS
LIN {X 0.120,Y -386.592,Z 1402.443,A 0.000,B 0.000,C 90.000,E1 79.746} C_DIS
LIN {X -0.025,Y -375.273,Z 1402.432,A 0.000,B 0.000,C 90.000,E1 77.757} C_DIS
LIN {X 0.044,Y -363.898,Z 1402.421,A 0.000,B 0.000,C 90.000,E1 75.700} C_DIS
LIN {X 0.008,Y -354.020,Z 1402.411,A 0.000,B 0.000,C 90.000,E1 73.921} C_DIS
LIN {X -0.110,Y -344.114,Z 1402.401,A 0.000,B 0.000,C 90.000,E1 72.127} C_DIS
LIN {X 0.115,Y -332.404,Z 1402.389,A 0.000,B 0.000,C 90.000,E1 69.934} C_DIS
LIN {X 0.039,Y -316.171,Z 1402.371,A 0.000,B 0.000,C 90.000,E1 66.794} C_DIS
LIN {X -0.016,Y -301.228,Z 1402.353,A 0.000,B 0.000,C 90.000,E1 63.563} C_DIS
LIN {X -0.104,Y -288.159,Z 1402.335,A 0.000,B 0.000,C 90.000,E1 60.255} C_DIS
LIN {X -0.016,Y -276.539,Z 1402.316,A 0.000,B 0.000,C 90.000,E1 56.834} C_DIS
LIN {X 0.033,Y -266.903,Z 1402.298,A 0.000,B 0.000,C 90.000,E1 53.703} C_DIS
LIN {X 0.025,Y -258.832,Z 1402.283,A 0.000,B 0.000,C 90.000,E1 50.884} C_DIS
LIN {X -0.037,Y -249.266,Z 1402.263,A 0.000,B 0.000,C 90.000,E1 47.310} C_DIS
LIN {X 0.099,Y -240.505,Z 1402.242,A 0.000,B 0.000,C 90.000,E1 43.623} C_DIS
LIN {X -0.013,Y -232.600,Z 1402.222,A 0.000,B 0.000,C 90.000,E1 39.930} C_DIS
LIN {X -0.086,Y -225.595,Z 1402.201,A 0.000,B 0.000,C 90.000,E1 36.171} C_DIS
LIN {X -0.088,Y -219.422,Z 1402.180,A 0.000,B 0.000,C 90.000,E1 32.339} C_DIS
LIN {X -0.003,Y -214.143,Z 1402.158,A 0.000,B 0.000,C 90.000,E1 28.437} C_DIS
LIN {X -0.009,Y -209.783,Z 1402.136,A 0.000,B 0.000,C 90.000,E1 24.515} C_DIS
LIN {X 0.003,Y -205.826,Z 1402.110,A 0.000,B 0.000,C 90.000,E1 19.758} C_DIS
LIN {X 0.048,Y -202.882,Z 1402.083,A 0.000,B 0.000,C 90.000,E1 14.954} C_DIS
LIN {X 0.004,Y -201.040,Z 1402.061,A 0.000,B 0.000,C 90.000,E1 10.950} C_DIS
LIN {X 0.095,Y -199.774,Z 1402.043,A 0.000,B 0.000,C 90.000,E1 7.701} C_DIS
LIN {X 0.058,Y -198.465,Z 1402.021,A 0.000,B 0.000,C 90.000,E1 3.669} C_DIS
LIN {X -0.036,Y -197.485,Z 1401.997,A 0.000,B 0.000,C 90.000,E1 359.542} C_DIS
LIN {X -0.042,Y -196.780,Z 1401.966,A 0.000,B 0.000,C 90.000,E1 353.856} C_DIS
LIN {X -0.099,Y -197.075,Z 1401.939,A 0.000,B 0.000,C 90.000,E1 348.993} C_DIS
LIN {X 0.078,Y -199.506,Z 1401.898,A 0.000,B 0.000,C 90.000,E1 341.638} C_DIS
LIN {X 0.083,Y -202.816,Z 1401.871,A 0.000,B 0.000,C 90.000,E1 336.794} C_DIS
LIN {X -0.031,Y -206.836,Z 1401.849,A 0.000,B 0.000,C 90.000,E1 332.820} C_DIS
LIN {X -0.100,Y -211.961,Z 1401.827,A 0.000,B 0.000,C 90.000,E1 328.869} C_DIS
LIN {X 0.094,Y -216.994,Z 1401.809,A 0.000,B 0.000,C 90.000,E1 325.674} C_DIS
LIN {X 0.131,Y -222.996,Z 1401.792,A 0.000,B 0.000,C 90.000,E1 322.557} C_DIS
LIN {X -0.080,Y -229.890,Z 1401.775,A 0.000,B 0.000,C 90.000,E1 319.542} C_DIS
LIN {X -0.045,Y -238.653,Z 1401.756,A 0.000,B 0.000,C 90.000,E1 316.134} C_DIS
LIN {X 0.094,Y -248.534,Z 1401.738,A 0.000,B 0.000,C 90.000,E1 312.771} C_DIS
LIN {X 0.011,Y -258.561,Z 1401.722,A 0.000,B 0.000,C 90.000,E1 309.886} C_DIS
LIN {X -0.084,Y -271.105,Z 1401.704,A 0.000,B 0.000,C 90.000,E1 306.710} C_DIS
LIN {X 0.061,Y -282.092,Z 1401.690,A 0.000,B 0.000,C 90.000,E1 304.246} C_DIS
LIN {X 0.032,Y -290.964,Z 1401.681,A 0.000,B 0.000,C 90.000,E1 302.546} C_DIS
LIN {X -0.014,Y -298.918,Z 1401.673,A 0.000,B 0.000,C 90.000,E1 301.209} C_DIS
LIN {X 0.071,Y -310.030,Z 1401.664,A 0.000,B 0.000,C 90.000,E1 299.539} C_DIS
LIN {X 0.099,Y -317.350,Z 1401.659,A 0.000,B 0.000,C 90.000,E1 298.565} C_DIS
LIN {X -0.007,Y -338.535,Z 1401.645,A 0.000,B 0.000,C 90.000,E1 296.155} C_DIS
LIN {X -0.045,Y -352.079,Z 1401.637,A 0.000,B 0.000,C 90.000,E1 294.719} C_DIS
LIN {X 0.077,Y -365.432,Z 1401.629,A 0.000,B 0.000,C 90.000,E1 293.281} C_DIS
LIN {X 0.069,Y -375.778,Z 1401.623,A 0.000,B 0.000,C 90.000,E1 292.153} C_DIS
LIN {X 0.001,Y -385.722,Z 1401.617,A 0.000,B 0.000,C 90.000,E1 291.046} C_DIS
LIN {X -0.106,Y -398.237,Z 1401.609,A 0.000,B 0.000,C 90.000,E1 289.631} C_DIS
LIN {X -0.084,Y -415.687,Z 1401.598,A 0.000,B 0.000,C 90.000,E1 287.692} C_DIS
LIN {X 0.000,Y -422.981,Z 1401.594,A 0.000,B 0.000,C 90.000,E1 286.858} C_DIS
LIN {X 0.158,Y -429.688,Z 1401.589,A 0.000,B 0.000,C 90.000,E1 286.024} C_DIS
LIN {X -0.044,Y -435.602,Z 1401.585,A 0.000,B 0.000,C 90.000,E1 285.245} C_DIS
LIN {X 0.119,Y -440.695,Z 1401.580,A 0.000,B 0.000,C 90.000,E1 284.426} C_DIS
LIN {X 0.007,Y -444.938,Z 1401.576,A 0.000,B 0.000,C 90.000,E1 283.647} C_DIS
LIN {X 0.028,Y -447.302,Z 1401.573,A 0.000,B 0.000,C 90.000,E1 283.119} C_DIS
LIN {X 0.064,Y -449.341,Z 1401.570,A 0.000,B 0.000,C 90.000,E1 282.591} C_DIS
LIN {X 0.107,Y -451.051,Z 1401.567,A 0.000,B 0.000,C 90.000,E1 282.063} C_DIS
LIN {X 0.161,Y -452.380,Z 1401.564,A 0.000,B 0.000,C 90.000,E1 281.535} C_DIS
LIN {X 0.225,Y -453.361,Z 1401.561,A 0.000,B 0.000,C 90.000,E1 281.007} C_DIS
LIN {X -0.234,Y -453.898,Z 1401.558,A 0.000,B 0.000,C 90.000,E1 280.546} C_DIS
LIN {X -0.159,Y -454.064,Z 1401.556,A 0.000,B 0.000,C 90.000,E1 280.018} C_DIS
LIN {X -0.158,Y -453.802,Z 1401.553,A 0.000,B 0.000,C 90.000,E1 279.500} C_DIS
LIN {X -0.082,Y -453.045,Z 1401.550,A 0.000,B 0.000,C 90.000,E1 278.973} C_DIS
LIN {X -0.078,Y -451.695,Z 1401.547,A 0.000,B 0.000,C 90.000,E1 278.454} C_DIS
LIN {X -0.076,Y -449.770,Z 1401.544,A 0.000,B 0.000,C 90.000,E1 277.936} C_DIS
LIN {X -0.022,Y -447.149,Z 1401.541,A 0.000,B 0.000,C 90.000,E1 277.409} C_DIS
LIN {X -0.046,Y -443.789,Z 1401.538,A 0.000,B 0.000,C 90.000,E1 276.891} C_DIS
LIN {X -0.087,Y -439.430,Z 1401.535,A 0.000,B 0.000,C 90.000,E1 276.372} C_DIS
LIN {X -0.147,Y -433.961,Z 1401.532,A 0.000,B 0.000,C 90.000,E1 275.853} C_DIS
LIN {X 0.105,Y -427.790,Z 1401.530,A 0.000,B 0.000,C 90.000,E1 275.334} C_DIS
LIN {X -0.040,Y -421.509,Z 1401.527,A 0.000,B 0.000,C 90.000,E1 274.935} C_DIS
LIN {X 0.185,Y -414.824,Z 1401.525,A 0.000,B 0.000,C 90.000,E1 274.531} C_DIS
LIN {X 0.145,Y -404.996,Z 1401.523,A 0.000,B 0.000,C 90.000,E1 274.073} C_DIS
LIN {X 0.106,Y -395.246,Z 1401.521,A 0.000,B 0.000,C 90.000,E1 273.669} C_DIS
LIN {X -0.024,Y -385.497,Z 1401.518,A 0.000,B 0.000,C 90.000,E1 273.326} C_DIS
LIN {X 0.111,Y -375.471,Z 1401.517,A 0.000,B 0.000,C 90.000,E1 272.980} C_DIS
LIN {X 0.183,Y -364.900,Z 1401.515,A 0.000,B 0.000,C 90.000,E1 272.694} C_DIS
LIN {X -0.173,Y -353.954,Z 1401.514,A 0.000,B 0.000,C 90.000,E1 272.522} C_DIS
LIN {X 0.158,Y -341.763,Z 1401.513,A 0.000,B 0.000,C 90.000,E1 272.293} C_DIS
LIN {X 0.139,Y -328.078,Z 1401.512,A 0.000,B 0.000,C 90.000,E1 272.178} C_DIS
LIN {X -0.078,Y -315.529,Z 1401.512,A 0.000,B 0.000,C 90.000,E1 272.178} C_DIS
LIN {X -0.071,Y -181.237,Z 1401.512,A 0.000,B 0.000,C 90.000,E1 272.178} C_DIS
LIN {X -0.090,Y -181.573,Z 1401.502,A 0.000,B 0.000,C 90.000,E1 270.458} C_DIS
LIN {X 0.068,Y -180.907,Z 1401.474,A 0.000,B 0.000,C 90.000,E1 265.355} C_DIS
LIN {X -0.038,Y -180.693,Z 1401.470,A 0.000,B 0.000,C 90.000,E1 264.546} C_DIS
LIN {X 0.041,Y -178.777,Z 1401.442,A 0.000,B 0.000,C 90.000,E1 259.454} C_DIS
LIN {X -0.057,Y -175.823,Z 1401.413,A 0.000,B 0.000,C 90.000,E1 254.393} C_DIS
LIN {X -0.057,Y -172.011,Z 1401.385,A 0.000,B 0.000,C 90.000,E1 249.263} C_DIS
LIN {X -0.080,Y -171.431,Z 1401.380,A 0.000,B 0.000,C 90.000,E1 248.411} C_DIS
LIN {X -0.025,Y -167.668,Z 1401.356,A 0.000,B 0.000,C 90.000,E1 244.076} C_DIS
LIN {X -0.084,Y -166.339,Z 1401.346,A 0.000,B 0.000,C 90.000,E1 242.359} C_DIS
LIN {X -0.091,Y -163.076,Z 1401.327,A 0.000,B 0.000,C 90.000,E1 238.869} C_DIS
LIN {X -0.040,Y -161.017,Z 1401.312,A 0.000,B 0.000,C 90.000,E1 236.215} C_DIS
LIN {X 0.069,Y -157.759,Z 1401.293,A 0.000,B 0.000,C 90.000,E1 232.637} C_DIS
LIN {X 0.008,Y -155.797,Z 1401.278,A 0.000,B 0.000,C 90.000,E1 229.989} C_DIS
LIN {X 0.062,Y -152.050,Z 1401.253,A 0.000,B 0.000,C 90.000,E1 225.486} C_DIS
LIN {X 0.079,Y -150.299,Z 1401.238,A 0.000,B 0.000,C 90.000,E1 222.771} C_DIS
LIN {X 0.005,Y -147.045,Z 1401.213,A 0.000,B 0.000,C 90.000,E1 218.257} C_DIS
LIN {X -0.002,Y -145.624,Z 1401.197,A 0.000,B 0.000,C 90.000,E1 215.518} C_DIS
LIN {X -0.004,Y -143.008,Z 1401.172,A 0.000,B 0.000,C 90.000,E1 210.924} C_DIS
LIN {X -0.073,Y -141.634,Z 1401.151,A 0.000,B 0.000,C 90.000,E1 207.257} C_DIS
LIN {X -0.021,Y -139.437,Z 1401.115,A 0.000,B 0.000,C 90.000,E1 200.737} C_DIS
LIN {X 0.032,Y -139.169,Z 1401.105,A 0.000,B 0.000,C 90.000,E1 198.852} C_DIS
LIN {X -0.071,Y -138.317,Z 1401.053,A 0.000,B 0.000,C 90.000,E1 189.557} C_DIS
LIN {X -0.062,Y -139.474,Z 1401.006,A 0.000,B 0.000,C 90.000,E1 181.146} C_DIS
LIN {X 0.019,Y -141.052,Z 1400.975,A 0.000,B 0.000,C 90.000,E1 175.527} C_DIS
LIN {X -0.027,Y -142.424,Z 1400.960,A 0.000,B 0.000,C 90.000,E1 172.761} C_DIS
LIN {X 0.033,Y -144.659,Z 1400.934,A 0.000,B 0.000,C 90.000,E1 168.117} C_DIS
LIN {X 0.017,Y -147.242,Z 1400.914,A 0.000,B 0.000,C 90.000,E1 164.448} C_DIS
LIN {X 0.036,Y -150.559,Z 1400.888,A 0.000,B 0.000,C 90.000,E1 159.880} C_DIS
LIN {X -0.026,Y -154.027,Z 1400.868,A 0.000,B 0.000,C 90.000,E1 156.282} C_DIS
LIN {X 0.043,Y -157.443,Z 1400.848,A 0.000,B 0.000,C 90.000,E1 152.666} C_DIS
LIN {X -0.008,Y -161.658,Z 1400.828,A 0.000,B 0.000,C 90.000,E1 149.125} C_DIS
LIN {X 0.010,Y -165.853,Z 1400.809,A 0.000,B 0.000,C 90.000,E1 145.595} C_DIS
LIN {X 0.001,Y -170.828,Z 1400.790,A 0.000,B 0.000,C 90.000,E1 142.110} C_DIS
LIN {X -0.083,Y -175.698,Z 1400.770,A 0.000,B 0.000,C 90.000,E1 138.690} C_DIS
LIN {X 0.040,Y -181.310,Z 1400.751,A 0.000,B 0.000,C 90.000,E1 135.243} C_DIS
LIN {X -0.089,Y -186.793,Z 1400.733,A 0.000,B 0.000,C 90.000,E1 131.919} C_DIS
LIN {X -0.018,Y -191.385,Z 1400.719,A 0.000,B 0.000,C 90.000,E1 129.402} C_DIS
LIN {X 0.065,Y -197.228,Z 1400.701,A 0.000,B 0.000,C 90.000,E1 126.091} C_DIS
LIN {X 0.023,Y -199.537,Z 1400.694,A 0.000,B 0.000,C 90.000,E1 124.945} C_DIS
LIN {X -0.003,Y -310.073,Z 1400.694,A 0.000,B 0.000,C 90.000,E1 124.945} C_DIS
LIN {X 0.132,Y -311.632,Z 1400.694,A 0.000,B 0.000,C 90.000,E1 124.898} C_DIS
LIN {X 0.058,Y -316.561,Z 1400.693,A 0.000,B 0.000,C 90.000,E1 124.692} C_DIS
LIN {X -0.017,Y -319.171,Z 1400.692,A 0.000,B 0.000,C 90.000,E1 124.485} C_DIS
LIN {X 0.004,Y -322.944,Z 1400.689,A 0.000,B 0.000,C 90.000,E1 123.992} C_DIS
LIN {X 0.082,Y -324.655,Z 1400.687,A 0.000,B 0.000,C 90.000,E1 123.658} C_DIS
LIN {X -0.012,Y -327.093,Z 1400.684,A 0.000,B 0.000,C 90.000,E1 123.038} C_DIS
LIN {X 0.023,Y -337.645,Z 1400.668,A 0.000,B 0.000,C 90.000,E1 120.207} C_DIS
LIN {X 0.012,Y -349.543,Z 1400.652,A 0.000,B 0.000,C 90.000,E1 117.436} C_DIS
LIN {X 0.008,Y -362.898,Z 1400.637,A 0.000,B 0.000,C 90.000,E1 114.719} C_DIS
LIN {X 0.146,Y -376.079,Z 1400.624,A 0.000,B 0.000,C 90.000,E1 112.333} C_DIS
LIN {X -0.171,Y -390.591,Z 1400.611,A 0.000,B 0.000,C 90.000,E1 110.066} C_DIS
LIN {X 0.111,Y -406.534,Z 1400.599,A 0.000,B 0.000,C 90.000,E1 107.764} C_DIS
LIN {X 0.166,Y -424.019,Z 1400.587,A 0.000,B 0.000,C 90.000,E1 105.552} C_DIS
LIN {X 0.137,Y -443.146,Z 1400.575,A 0.000,B 0.000,C 90.000,E1 103.411} C_DIS
LIN {X 0.006,Y -463.223,Z 1400.563,A 0.000,B 0.000,C 90.000,E1 101.422} C_DIS
LIN {X 0.198,Y -483.821,Z 1400.553,A 0.000,B 0.000,C 90.000,E1 99.557} C_DIS
LIN {X -0.170,Y -485.944,Z 1400.552,A 0.000,B 0.000,C 90.000,E1 99.378} C_DIS
LIN {X -0.139,Y -487.561,Z 1400.551,A 0.000,B 0.000,C 90.000,E1 99.151} C_DIS
LIN {X 0.238,Y -488.931,Z 1400.549,A 0.000,B 0.000,C 90.000,E1 98.859} C_DIS
LIN {X 0.132,Y -489.944,Z 1400.548,A 0.000,B 0.000,C 90.000,E1 98.624} C_DIS
LIN {X -0.140,Y -491.091,Z 1400.545,A 0.000,B 0.000,C 90.000,E1 98.163} C_DIS
LIN {X 0.082,Y -491.221,Z 1400.542,A 0.000,B 0.000,C 90.000,E1 97.644} C_DIS
LIN {X -0.175,Y -490.356,Z 1400.540,A 0.000,B 0.000,C 90.000,E1 97.182} C_DIS
LIN {X 0.056,Y -488.349,Z 1400.537,A 0.000,B 0.000,C 90.000,E1 96.663} C_DIS
LIN {X 0.001,Y -481.710,Z 1400.532,A 0.000,B 0.000,C 90.000,E1 95.682} C_DIS
LIN {X 0.159,Y -465.602,Z 1400.518,A 0.000,B 0.000,C 90.000,E1 93.154} C_DIS
LIN {X 0.053,Y -457.228,Z 1400.510,A 0.000,B 0.000,C 90.000,E1 91.892} C_DIS
LIN {X 0.111,Y -439.363,Z 1400.495,A 0.000,B 0.000,C 90.000,E1 89.026} C_DIS
LIN {X 0.077,Y -427.231,Z 1400.483,A 0.000,B 0.000,C 90.000,E1 86.906} C_DIS
LIN {X 0.132,Y -416.449,Z 1400.472,A 0.000,B 0.000,C 90.000,E1 85.008} C_DIS
LIN {X -0.026,Y -405.502,Z 1400.462,A 0.000,B 0.000,C 90.000,E1 83.109} C_DIS
LIN {X 0.013,Y -396.028,Z 1400.452,A 0.000,B 0.000,C 90.000,E1 81.432} C_DIS
LIN {X -0.055,Y -386.414,Z 1400.443,A 0.000,B 0.000,C 90.000,E1 79.746} C_DIS
LIN {X 0.167,Y -375.088,Z 1400.432,A 0.000,B 0.000,C 90.000,E1 77.701} C_DIS
LIN {X -0.129,Y -363.708,Z 1400.420,A 0.000,B 0.000,C 90.000,E1 75.700} C_DIS
LIN {X -0.165,Y -353.821,Z 1400.411,A 0.000,B 0.000,C 90.000,E1 73.921} C_DIS
LIN {X 0.153,Y -343.894,Z 1400.400,A 0.000,B 0.000,C 90.000,E1 72.054} C_DIS
LIN {X -0.055,Y -332.177,Z 1400.388,A 0.000,B 0.000,C 90.000,E1 69.934} C_DIS
LIN {X 0.097,Y -314.395,Z 1400.369,A 0.000,B 0.000,C 90.000,E1 66.433} C_DIS
LIN {X 0.086,Y -301.042,Z 1400.353,A 0.000,B 0.000,C 90.000,E1 63.512} C_DIS
LIN {X -0.019,Y -288.002,Z 1400.334,A 0.000,B 0.000,C 90.000,E1 60.205} C_DIS
LIN {X 0.103,Y -277.511,Z 1400.318,A 0.000,B 0.000,C 90.000,E1 57.120} C_DIS
LIN {X -0.126,Y -268.916,Z 1400.302,A 0.000,B 0.000,C 90.000,E1 54.402} C_DIS
LIN {X 0.131,Y -260.783,Z 1400.286,A 0.000,B 0.000,C 90.000,E1 51.537} C_DIS
LIN {X -0.039,Y -251.108,Z 1400.267,A 0.000,B 0.000,C 90.000,E1 48.000} C_DIS
LIN {X -0.011,Y -242.192,Z 1400.246,A 0.000,B 0.000,C 90.000,E1 44.352} C_DIS
LIN {X 0.092,Y -234.144,Z 1400.226,A 0.000,B 0.000,C 90.000,E1 40.620} C_DIS
LIN {X 0.024,Y -226.989,Z 1400.205,A 0.000,B 0.000,C 90.000,E1 36.870} C_DIS
LIN {X 0.063,Y -220.664,Z 1400.184,A 0.000,B 0.000,C 90.000,E1 33.038} C_DIS
LIN {X -0.079,Y -215.258,Z 1400.162,A 0.000,B 0.000,C 90.000,E1 29.205} C_DIS
LIN {X -0.050,Y -210.759,Z 1400.140,A 0.000,B 0.000,C 90.000,E1 25.283} C_DIS
LIN {X -0.037,Y -206.621,Z 1400.114,A 0.000,B 0.000,C 90.000,E1 20.536} C_DIS
LIN {X 0.033,Y -203.621,Z 1400.087,A 0.000,B 0.000,C 90.000,E1 15.733} C_DIS
LIN {X 0.065,Y -201.692,Z 1400.065,A 0.000,B 0.000,C 90.000,E1 11.715} C_DIS
LIN {X 0.024,Y -200.080,Z 1400.043,A 0.000,B 0.000,C 90.000,E1 7.701} C_DIS
LIN {X -0.004,Y -198.771,Z 1400.020,A 0.000,B 0.000,C 90.000,E1 3.669} C_DIS
LIN {X -0.036,Y -197.754,Z 1399.997,A 0.000,B 0.000,C 90.000,E1 359.542} C_DIS
LIN {X -0.020,Y -197.064,Z 1399.970,A 0.000,B 0.000,C 90.000,E1 354.666} C_DIS
LIN {X -0.079,Y -197.300,Z 1399.939,A 0.000,B 0.000,C 90.000,E1 348.993} C_DIS
LIN {X 0.110,Y -199.734,Z 1399.898,A 0.000,B 0.000,C 90.000,E1 341.638} C_DIS
LIN {X -0.062,Y -203.030,Z 1399.871,A 0.000,B 0.000,C 90.000,E1 336.847} C_DIS
LIN {X 0.019,Y -207.051,Z 1399.849,A 0.000,B 0.000,C 90.000,E1 332.820} C_DIS
LIN {X -0.042,Y -212.177,Z 1399.827,A 0.000,B 0.000,C 90.000,E1 328.869} C_DIS
LIN {X -0.148,Y -218.586,Z 1399.805,A 0.000,B 0.000,C 90.000,E1 324.975} C_DIS
LIN {X 0.059,Y -224.815,Z 1399.788,A 0.000,B 0.000,C 90.000,E1 321.823} C_DIS
LIN {X 0.042,Y -231.933,Z 1399.771,A 0.000,B 0.000,C 90.000,E1 318.771} C_DIS
LIN {X -0.026,Y -240.885,Z 1399.752,A 0.000,B 0.000,C 90.000,E1 315.405} C_DIS
LIN {X 0.011,Y -251.043,Z 1399.734,A 0.000,B 0.000,C 90.000,E1 312.081} C_DIS
LIN {X 0.036,Y -262.701,Z 1399.716,A 0.000,B 0.000,C 90.000,E1 308.830} C_DIS
LIN {X 0.022,Y -274.209,Z 1399.700,A 0.000,B 0.000,C 90.000,E1 306.011} C_DIS
LIN {X 0.132,Y -283.837,Z 1399.689,A 0.000,B 0.000,C 90.000,E1 303.913} C_DIS
LIN {X 0.130,Y -292.903,Z 1399.679,A 0.000,B 0.000,C 90.000,E1 302.212} C_DIS
LIN {X 0.114,Y -301.101,Z 1399.672,A 0.000,B 0.000,C 90.000,E1 300.875} C_DIS
LIN {X -0.181,Y -312.417,Z 1399.662,A 0.000,B 0.000,C 90.000,E1 299.283} C_DIS
LIN {X 0.038,Y -319.955,Z 1399.657,A 0.000,B 0.000,C 90.000,E1 298.281} C_DIS
LIN {X 0.144,Y -343.767,Z 1399.642,A 0.000,B 0.000,C 90.000,E1 295.591} C_DIS
LIN {X -0.180,Y -357.254,Z 1399.634,A 0.000,B 0.000,C 90.000,E1 294.207} C_DIS
LIN {X -0.006,Y -367.570,Z 1399.628,A 0.000,B 0.000,C 90.000,E1 293.078} C_DIS
LIN {X -0.060,Y -377.901,Z 1399.622,A 0.000,B 0.000,C 90.000,E1 291.950} C_DIS
LIN {X -0.169,Y -390.320,Z 1399.614,A 0.000,B 0.000,C 90.000,E1 290.556} C_DIS
LIN {X -0.149,Y -405.259,Z 1399.605,A 0.000,B 0.000,C 90.000,E1 288.852} C_DIS
LIN {X -0.018,Y -417.824,Z 1399.597,A 0.000,B 0.000,C 90.000,E1 287.457} C_DIS
LIN {X 0.091,Y -424.965,Z 1399.592,A 0.000,B 0.000,C 90.000,E1 286.622} C_DIS
LIN {X -0.153,Y -431.517,Z 1399.588,A 0.000,B 0.000,C 90.000,E1 285.843} C_DIS
LIN {X 0.083,Y -437.185,Z 1399.583,A 0.000,B 0.000,C 90.000,E1 285.009} C_DIS
LIN {X 0.054,Y -440.577,Z 1399.580,A 0.000,B 0.000,C 90.000,E1 284.481} C_DIS
LIN {X -0.061,Y -444.871,Z 1399.576,A 0.000,B 0.000,C 90.000,E1 283.703} C_DIS
LIN {X 0.193,Y -448.319,Z 1399.572,A 0.000,B 0.000,C 90.000,E1 282.883} C_DIS
LIN {X 0.040,Y -451.079,Z 1399.567,A 0.000,B 0.000,C 90.000,E1 282.119} C_DIS
LIN {X 0.093,Y -452.453,Z 1399.564,A 0.000,B 0.000,C 90.000,E1 281.591} C_DIS
LIN {X 0.070,Y -453.479,Z 1399.562,A 0.000,B 0.000,C 90.000,E1 281.074} C_DIS
LIN {X 0.143,Y -454.061,Z 1399.559,A 0.000,B 0.000,C 90.000,E1 280.546} C_DIS
LIN {X 0.219,Y -454.280,Z 1399.556,A 0.000,B 0.000,C 90.000,E1 280.018} C_DIS
LIN {X -0.227,Y -454.064,Z 1399.553,A 0.000,B 0.000,C 90.000,E1 279.557} C_DIS
LIN {X -0.150,Y -453.341,Z 1399.550,A 0.000,B 0.000,C 90.000,E1 279.029} C_DIS
LIN {X -0.145,Y -452.097,Z 1399.547,A 0.000,B 0.000,C 90.000,E1 278.511} C_DIS
LIN {X -0.142,Y -450.276,Z 1399.544,A 0.000,B 0.000,C 90.000,E1 277.992} C_DIS
LIN {X -0.086,Y -447.777,Z 1399.541,A 0.000,B 0.000,C 90.000,E1 277.466} C_DIS
LIN {X -0.107,Y -444.540,Z 1399.539,A 0.000,B 0.000,C 90.000,E1 276.947} C_DIS
LIN {X -0.143,Y -440.331,Z 1399.536,A 0.000,B 0.000,C 90.000,E1 276.429} C_DIS
LIN {X -0.200,Y -435.036,Z 1399.533,A 0.000,B 0.000,C 90.000,E1 275.910} C_DIS
LIN {X 0.010,Y -429.028,Z 1399.530,A 0.000,B 0.000,C 90.000,E1 275.391} C_DIS
LIN {X 0.197,Y -422.751,Z 1399.528,A 0.000,B 0.000,C 90.000,E1 274.935} C_DIS
LIN {X -0.084,Y -415.974,Z 1399.525,A 0.000,B 0.000,C 90.000,E1 274.588} C_DIS
LIN {X 0.047,Y -409.384,Z 1399.524,A 0.000,B 0.000,C 90.000,E1 274.245} C_DIS
LIN {X -0.125,Y -399.613,Z 1399.521,A 0.000,B 0.000,C 90.000,E1 273.841} C_DIS
LIN {X -0.041,Y -389.658,Z 1399.519,A 0.000,B 0.000,C 90.000,E1 273.440} C_DIS
LIN {X 0.003,Y -379.777,Z 1399.517,A 0.000,B 0.000,C 90.000,E1 273.094} C_DIS
LIN {X -0.115,Y -369.027,Z 1399.516,A 0.000,B 0.000,C 90.000,E1 272.808} C_DIS
LIN {X -0.167,Y -358.478,Z 1399.514,A 0.000,B 0.000,C 90.000,E1 272.579} C_DIS
LIN {X 0.069,Y -351.057,Z 1399.513,A 0.000,B 0.000,C 90.000,E1 272.407} C_DIS
LIN {X 0.119,Y -337.547,Z 1399.513,A 0.000,B 0.000,C 90.000,E1 272.236} C_DIS
LIN {X -0.057,Y -323.581,Z 1399.512,A 0.000,B 0.000,C 90.000,E1 272.178} C_DIS
LIN {X -0.102,Y -320.692,Z 1399.512,A 0.000,B 0.000,C 90.000,E1 272.178} C_DIS
LIN {X -0.083,Y -181.238,Z 1399.512,A 0.000,B 0.000,C 90.000,E1 272.178} C_DIS
LIN {X 0.055,Y -181.574,Z 1399.502,A 0.000,B 0.000,C 90.000,E1 270.401} C_DIS
LIN {X 0.032,Y -180.905,Z 1399.474,A 0.000,B 0.000,C 90.000,E1 265.355} C_DIS
LIN {X -0.074,Y -180.687,Z 1399.470,A 0.000,B 0.000,C 90.000,E1 264.546} C_DIS
LIN {X 0.004,Y -178.771,Z 1399.441,A 0.000,B 0.000,C 90.000,E1 259.454} C_DIS
LIN {X 0.076,Y -175.816,Z 1399.413,A 0.000,B 0.000,C 90.000,E1 254.338} C_DIS
LIN {X 0.069,Y -172.004,Z 1399.385,A 0.000,B 0.000,C 90.000,E1 249.209} C_DIS
LIN {X 0.044,Y -171.421,Z 1399.380,A 0.000,B 0.000,C 90.000,E1 248.358} C_DIS
LIN {X 0.091,Y -167.658,Z 1399.356,A 0.000,B 0.000,C 90.000,E1 244.024} C_DIS
LIN {X 0.028,Y -166.326,Z 1399.346,A 0.000,B 0.000,C 90.000,E1 242.308} C_DIS
LIN {X 0.014,Y -163.066,Z 1399.327,A 0.000,B 0.000,C 90.000,E1 238.820} C_DIS
LIN {X -0.075,Y -161.004,Z 1399.312,A 0.000,B 0.000,C 90.000,E1 236.215} C_DIS
LIN {X 0.036,Y -157.748,Z 1399.292,A 0.000,B 0.000,C 90.000,E1 232.637} C_DIS
LIN {X -0.026,Y -155.787,Z 1399.278,A 0.000,B 0.000,C 90.000,E1 229.989} C_DIS
LIN {X 0.029,Y -152.041,Z 1399.253,A 0.000,B 0.000,C 90.000,E1 225.486} C_DIS
LIN {X 0.047,Y -150.289,Z 1399.238,A 0.000,B 0.000,C 90.000,E1 222.771} C_DIS
LIN {X -0.027,Y -147.038,Z 1399.213,A 0.000,B 0.000,C 90.000,E1 218.257} C_DIS
LIN {X -0.035,Y -145.618,Z 1399.197,A 0.000,B 0.000,C 90.000,E1 215.518} C_DIS
LIN {X -0.036,Y -143.002,Z 1399.172,A 0.000,B 0.000,C 90.000,E1 210.924} C_DIS
LIN {X 0.022,Y -141.630,Z 1399.151,A 0.000,B 0.000,C 90.000,E1 207.206} C_DIS
LIN {X -0.053,Y -139.435,Z 1399.115,A 0.000,B 0.000,C 90.000,E1 200.737} C_DIS
LIN {X 0.001,Y -139.165,Z 1399.105,A 0.000,B 0.000,C 90.000,E1 198.852} C_DIS
LIN {X 0.035,Y -138.316,Z 1399.053,A 0.000,B 0.000,C 90.000,E1 189.500} C_DIS
LIN {X 0.046,Y -139.476,Z 1399.006,A 0.000,B 0.000,C 90.000,E1 181.088} C_DIS
LIN {X -0.013,Y -141.057,Z 1398.975,A 0.000,B 0.000,C 90.000,E1 175.527} C_DIS
LIN {X -0.060,Y -142.430,Z 1398.960,A 0.000,B 0.000,C 90.000,E1 172.761} C_DIS
LIN {X 0.001,Y -144.667,Z 1398.934,A 0.000,B 0.000,C 90.000,E1 168.117} C_DIS
LIN {X -0.015,Y -147.252,Z 1398.914,A 0.000,B 0.000,C 90.000,E1 164.448} C_DIS
LIN {X 0.002,Y -150.569,Z 1398.888,A 0.000,B 0.000,C 90.000,E1 159.880} C_DIS
LIN {X 0.082,Y -154.038,Z 1398.868,A 0.000,B 0.000,C 90.000,E1 156.230} C_DIS
LIN {X 0.009,Y -157.456,Z 1398.848,A 0.000,B 0.000,C 90.000,E1 152.666} C_DIS
LIN {X -0.042,Y -161.674,Z 1398.828,A 0.000,B 0.000,C 90.000,E1 149.125} C_DIS
LIN {X -0.025,Y -165.869,Z 1398.809,A 0.000,B 0.000,C 90.000,E1 145.595} C_DIS
LIN {X -0.034,Y -170.847,Z 1398.789,A 0.000,B 0.000,C 90.000,E1 142.110} C_DIS
LIN {X 0.013,Y -175.716,Z 1398.770,A 0.000,B 0.000,C 90.000,E1 138.647} C_DIS
LIN {X 0.003,Y -181.327,Z 1398.751,A 0.000,B 0.000,C 90.000,E1 135.243} C_DIS
LIN {X -0.001,Y -186.814,Z 1398.733,A 0.000,B 0.000,C 90.000,E1 131.881} C_DIS
LIN {X -0.056,Y -191.403,Z 1398.719,A 0.000,B 0.000,C 90.000,E1 129.402} C_DIS
LIN {X 0.027,Y -197.249,Z 1398.701,A 0.000,B 0.000,C 90.000,E1 126.091} C_DIS
LIN {X -0.038,Y -199.506,Z 1398.694,A 0.000,B 0.000,C 90.000,E1 124.978} C_DIS
LIN {X 0.083,Y -309.725,Z 1398.694,A 0.000,B 0.000,C 90.000,E1 124.945} C_DIS
LIN {X 0.073,Y -312.545,Z 1398.694,A 0.000,B 0.000,C 90.000,E1 124.898} C_DIS
LIN {X -0.002,Y -316.848,Z 1398.693,A 0.000,B 0.000,C 90.000,E1 124.692} C_DIS
LIN {X -0.080,Y -319.352,Z 1398.692,A 0.000,B 0.000,C 90.000,E1 124.485} C_DIS
LIN {X -0.156,Y -323.129,Z 1398.689,A 0.000,B 0.000,C 90.000,E1 123.992} C_DIS
LIN {X -0.077,Y -324.783,Z 1398.687,A 0.000,B 0.000,C 90.000,E1 123.658} C_DIS
LIN {X 0.007,Y -327.169,Z 1398.683,A 0.000,B 0.000,C 90.000,E1 123.007} C_DIS
LIN {X -0.140,Y -337.734,Z 1398.668,A 0.000,B 0.000,C 90.000,E1 120.207} C_DIS
LIN {X 0.157,Y -349.646,Z 1398.652,A 0.000,B 0.000,C 90.000,E1 117.385} C_DIS
LIN {X -0.010,Y -363.014,Z 1398.637,A 0.000,B 0.000,C 90.000,E1 114.695} C_DIS
LIN {X -0.026,Y -376.210,Z 1398.624,A 0.000,B 0.000,C 90.000,E1 112.333} C_DIS
LIN {X 0.155,Y -390.737,Z 1398.611,A 0.000,B 0.000,C 90.000,E1 109.993} C_DIS
LIN {X -0.068,Y -406.696,Z 1398.599,A 0.000,B 0.000,C 90.000,E1 107.764} C_DIS
LIN {X -0.016,Y -424.199,Z 1398.586,A 0.000,B 0.000,C 90.000,E1 105.552} C_DIS
LIN {X -0.046,Y -443.342,Z 1398.574,A 0.000,B 0.000,C 90.000,E1 103.411} C_DIS
LIN {X -0.171,Y -463.426,Z 1398.563,A 0.000,B 0.000,C 90.000,E1 101.422} C_DIS
LIN {X 0.029,Y -483.999,Z 1398.553,A 0.000,B 0.000,C 90.000,E1 99.557} C_DIS
LIN {X 0.126,Y -486.051,Z 1398.552,A 0.000,B 0.000,C 90.000,E1 99.321} C_DIS
LIN {X 0.145,Y -487.616,Z 1398.551,A 0.000,B 0.000,C 90.000,E1 99.095} C_DIS
LIN {X 0.040,Y -488.934,Z 1398.549,A 0.000,B 0.000,C 90.000,E1 98.859} C_DIS
LIN {X -0.066,Y -489.902,Z 1398.548,A 0.000,B 0.000,C 90.000,E1 98.624} C_DIS
LIN {X 0.148,Y -490.978,Z 1398.545,A 0.000,B 0.000,C 90.000,E1 98.106} C_DIS
LIN {X -0.117,Y -491.043,Z 1398.542,A 0.000,B 0.000,C 90.000,E1 97.644} C_DIS
LIN {X 0.112,Y -490.109,Z 1398.540,A 0.000,B 0.000,C 90.000,E1 97.125} C_DIS
LIN {X -0.144,Y -488.013,Z 1398.537,A 0.000,B 0.000,C 90.000,E1 96.663} C_DIS
LIN {X -0.115,Y -468.420,Z 1398.520,A 0.000,B 0.000,C 90.000,E1 93.669} C_DIS
LIN {X -0.181,Y -460.214,Z 1398.513,A 0.000,B 0.000,C 90.000,E1 92.407} C_DIS
LIN {X 0.159,Y -440.543,Z 1398.496,A 0.000,B 0.000,C 90.000,E1 89.255} C_DIS
LIN {X 0.153,Y -428.414,Z 1398.484,A 0.000,B 0.000,C 90.000,E1 87.135} C_DIS
LIN {X -0.214,Y -417.699,Z 1398.474,A 0.000,B 0.000,C 90.000,E1 85.298} C_DIS
LIN {X -0.002,Y -408.366,Z 1398.465,A 0.000,B 0.000,C 90.000,E1 83.628} C_DIS
LIN {X 0.168,Y -397.363,Z 1398.454,A 0.000,B 0.000,C 90.000,E1 81.659} C_DIS
LIN {X 0.059,Y -387.799,Z 1398.444,A 0.000,B 0.000,C 90.000,E1 79.982} C_DIS
LIN {X -0.045,Y -374.860,Z 1398.432,A 0.000,B 0.000,C 90.000,E1 77.701} C_DIS
LIN {X 0.031,Y -365.116,Z 1398.422,A 0.000,B 0.000,C 90.000,E1 75.936} C_DIS
LIN {X 0.018,Y -355.245,Z 1398.412,A 0.000,B 0.000,C 90.000,E1 74.157} C_DIS
LIN {X -0.076,Y -345.304,Z 1398.402,A 0.000,B 0.000,C 90.000,E1 72.362} C_DIS
LIN {X 0.069,Y -333.593,Z 1398.390,A 0.000,B 0.000,C 90.000,E1 70.188} C_DIS
LIN {X 0.023,Y -317.259,Z 1398.373,A 0.000,B 0.000,C 90.000,E1 67.050} C_DIS
LIN {X -0.003,Y -302.234,Z 1398.354,A 0.000,B 0.000,C 90.000,E1 63.819} C_DIS
LIN {X -0.055,Y -290.300,Z 1398.338,A 0.000,B 0.000,C 90.000,E1 60.845} C_DIS
LIN {X -0.049,Y -278.481,Z 1398.319,A 0.000,B 0.000,C 90.000,E1 57.454} C_DIS
LIN {X 0.057,Y -268.824,Z 1398.302,A 0.000,B 0.000,C 90.000,E1 54.322} C_DIS
LIN {X 0.051,Y -258.739,Z 1398.282,A 0.000,B 0.000,C 90.000,E1 50.803} C_DIS
LIN {X -0.012,Y -249.231,Z 1398.262,A 0.000,B 0.000,C 90.000,E1 47.229} C_DIS
LIN {X 0.122,Y -240.530,Z 1398.242,A 0.000,B 0.000,C 90.000,E1 43.542} C_DIS
LIN {X 0.009,Y -232.659,Z 1398.221,A 0.000,B 0.000,C 90.000,E1 39.850} C_DIS
LIN {X -0.065,Y -225.728,Z 1398.200,A 0.000,B 0.000,C 90.000,E1 36.091} C_DIS
LIN {X -0.066,Y -219.600,Z 1398.179,A 0.000,B 0.000,C 90.000,E1 32.260} C_DIS
LIN {X 0.018,Y -214.426,Z 1398.158,A 0.000,B 0.000,C 90.000,E1 28.359} C_DIS
LIN {X -0.072,Y -210.158,Z 1398.136,A 0.000,B 0.000,C 90.000,E1 24.463} C_DIS
LIN {X 0.033,Y -206.299,Z 1398.109,A 0.000,B 0.000,C 90.000,E1 19.685} C_DIS
LIN {X -0.036,Y -203.906,Z 1398.087,A 0.000,B 0.000,C 90.000,E1 15.717} C_DIS
LIN {X -0.048,Y -201.996,Z 1398.065,A 0.000,B 0.000,C 90.000,E1 11.715} C_DIS
LIN {X -0.080,Y -200.368,Z 1398.043,A 0.000,B 0.000,C 90.000,E1 7.701} C_DIS
LIN {X -0.097,Y -199.069,Z 1398.020,A 0.000,B 0.000,C 90.000,E1 3.669} C_DIS
LIN {X -0.036,Y -198.018,Z 1397.997,A 0.000,B 0.000,C 90.000,E1 359.542} C_DIS
LIN {X -0.011,Y -197.307,Z 1397.970,A 0.000,B 0.000,C 90.000,E1 354.666} C_DIS
LIN {X -0.059,Y -197.525,Z 1397.939,A 0.000,B 0.000,C 90.000,E1 348.993} C_DIS
LIN {X -0.046,Y -199.962,Z 1397.898,A 0.000,B 0.000,C 90.000,E1 341.692} C_DIS
LIN {X -0.019,Y -203.251,Z 1397.871,A 0.000,B 0.000,C 90.000,E1 336.847} C_DIS
LIN {X -0.116,Y -207.272,Z 1397.849,A 0.000,B 0.000,C 90.000,E1 332.871} C_DIS
LIN {X 0.016,Y -212.393,Z 1397.827,A 0.000,B 0.000,C 90.000,E1 328.869} C_DIS
LIN {X -0.081,Y -218.795,Z 1397.805,A 0.000,B 0.000,C 90.000,E1 324.975} C_DIS
LIN {X 0.132,Y -225.004,Z 1397.788,A 0.000,B 0.000,C 90.000,E1 321.823} C_DIS
LIN {X 0.123,Y -232.111,Z 1397.771,A 0.000,B 0.000,C 90.000,E1 318.771} C_DIS
LIN {X 0.064,Y -241.046,Z 1397.752,A 0.000,B 0.000,C 90.000,E1 315.405} C_DIS
LIN {X 0.108,Y -251.161,Z 1397.734,A 0.000,B 0.000,C 90.000,E1 312.081} C_DIS
LIN {X 0.141,Y -262.802,Z 1397.716,A 0.000,B 0.000,C 90.000,E1 308.830} C_DIS
LIN {X 0.057,Y -275.828,Z 1397.698,A 0.000,B 0.000,C 90.000,E1 305.678} C_DIS
LIN {X -0.145,Y -283.905,Z 1397.689,A 0.000,B 0.000,C 90.000,E1 303.992} C_DIS
LIN {X 0.005,Y -292.965,Z 1397.679,A 0.000,B 0.000,C 90.000,E1 302.260} C_DIS
LIN {X -0.019,Y -301.150,Z 1397.672,A 0.000,B 0.000,C 90.000,E1 300.924} C_DIS
LIN {X -0.091,Y -310.057,Z 1397.664,A 0.000,B 0.000,C 90.000,E1 299.617} C_DIS
LIN {X -0.048,Y -317.171,Z 1397.659,A 0.000,B 0.000,C 90.000,E1 298.665} C_DIS
LIN {X 0.087,Y -332.714,Z 1397.649,A 0.000,B 0.000,C 90.000,E1 296.821} C_DIS
LIN {X 0.044,Y -348.928,Z 1397.639,A 0.000,B 0.000,C 90.000,E1 295.079} C_DIS
LIN {X 0.060,Y -364.737,Z 1397.630,A 0.000,B 0.000,C 90.000,E1 293.387} C_DIS
LIN {X -0.098,Y -375.084,Z 1397.624,A 0.000,B 0.000,C 90.000,E1 292.280} C_DIS
LIN {X -0.033,Y -385.007,Z 1397.617,A 0.000,B 0.000,C 90.000,E1 291.153} C_DIS
LIN {X -0.052,Y -397.236,Z 1397.610,A 0.000,B 0.000,C 90.000,E1 289.758} C_DIS
LIN {X 0.093,Y -417.143,Z 1397.597,A 0.000,B 0.000,C 90.000,E1 287.528} C_DIS
LIN {X -0.060,Y -424.287,Z 1397.593,A 0.000,B 0.000,C 90.000,E1 286.732} C_DIS
LIN {X 0.100,Y -430.892,Z 1397.588,A 0.000,B 0.000,C 90.000,E1 285.898} C_DIS
LIN {X 0.030,Y -434.894,Z 1397.585,A 0.000,B 0.000,C 90.000,E1 285.371} C_DIS
LIN {X -0.127,Y -440.138,Z 1397.581,A 0.000,B 0.000,C 90.000,E1 284.592} C_DIS
LIN {X 0.077,Y -444.596,Z 1397.577,A 0.000,B 0.000,C 90.000,E1 283.772} C_DIS
LIN {X -0.104,Y -448.163,Z 1397.572,A 0.000,B 0.000,C 90.000,E1 283.008} C_DIS
LIN {X -0.256,Y -450.937,Z 1397.568,A 0.000,B 0.000,C 90.000,E1 282.243} C_DIS
LIN {X -0.202,Y -452.420,Z 1397.565,A 0.000,B 0.000,C 90.000,E1 281.715} C_DIS
LIN {X -0.138,Y -453.531,Z 1397.562,A 0.000,B 0.000,C 90.000,E1 281.186} C_DIS
LIN {X -0.067,Y -454.219,Z 1397.559,A 0.000,B 0.000,C 90.000,E1 280.658} C_DIS
LIN {X -0.071,Y -454.469,Z 1397.556,A 0.000,B 0.000,C 90.000,E1 280.141} C_DIS
LIN {X 0.009,Y -454.346,Z 1397.553,A 0.000,B 0.000,C 90.000,E1 279.613} C_DIS
LIN {X 0.016,Y -453.719,Z 1397.551,A 0.000,B 0.000,C 90.000,E1 279.095} C_DIS
LIN {X 0.092,Y -452.586,Z 1397.548,A 0.000,B 0.000,C 90.000,E1 278.568} C_DIS
LIN {X 0.096,Y -450.884,Z 1397.545,A 0.000,B 0.000,C 90.000,E1 278.049} C_DIS
LIN {X 0.095,Y -448.574,Z 1397.542,A 0.000,B 0.000,C 90.000,E1 277.530} C_DIS
LIN {X -0.106,Y -447.157,Z 1397.540,A 0.000,B 0.000,C 90.000,E1 277.296} C_DIS
LIN {X -0.130,Y -443.669,Z 1397.538,A 0.000,B 0.000,C 90.000,E1 276.777} C_DIS
LIN {X -0.168,Y -439.195,Z 1397.535,A 0.000,B 0.000,C 90.000,E1 276.258} C_DIS
LIN {X -0.128,Y -433.765,Z 1397.532,A 0.000,B 0.000,C 90.000,E1 275.739} C_DIS
LIN {X 0.216,Y -427.668,Z 1397.529,A 0.000,B 0.000,C 90.000,E1 275.220} C_DIS
LIN {X 0.069,Y -421.252,Z 1397.527,A 0.000,B 0.000,C 90.000,E1 274.821} C_DIS
LIN {X -0.076,Y -414.580,Z 1397.525,A 0.000,B 0.000,C 90.000,E1 274.473} C_DIS
LIN {X -0.118,Y -404.658,Z 1397.522,A 0.000,B 0.000,C 90.000,E1 274.012} C_DIS
LIN {X -0.115,Y -394.928,Z 1397.520,A 0.000,B 0.000,C 90.000,E1 273.612} C_DIS
LIN {X 0.159,Y -385.056,Z 1397.518,A 0.000,B 0.000,C 90.000,E1 273.212} C_DIS
LIN {X -0.043,Y -375.081,Z 1397.516,A 0.000,B 0.000,C 90.000,E1 272.922} C_DIS
LIN {X 0.083,Y -364.245,Z 1397.515,A 0.000,B 0.000,C 90.000,E1 272.636} C_DIS
LIN {X -0.158,Y -353.786,Z 1397.514,A 0.000,B 0.000,C 90.000,E1 272.465} C_DIS
LIN {X 0.154,Y -345.199,Z 1397.513,A 0.000,B 0.000,C 90.000,E1 272.293} C_DIS
LIN {X -0.085,Y -335.204,Z 1397.512,A 0.000,B 0.000,C 90.000,E1 272.236} C_DIS
LIN {X -0.161,Y -322.128,Z 1397.512,A 0.000,B 0.000,C 90.000,E1 272.178} C_DIS
LIN {X 0.062,Y -181.239,Z 1397.512,A 0.000,B 0.000,C 90.000,E1 272.121} C_DIS
LIN {X 0.059,Y -181.574,Z 1397.502,A 0.000,B 0.000,C 90.000,E1 270.401} C_DIS
LIN {X 0.036,Y -180.906,Z 1397.474,A 0.000,B 0.000,C 90.000,E1 265.355} C_DIS
LIN {X -0.071,Y -180.688,Z 1397.470,A 0.000,B 0.000,C 90.000,E1 264.546} C_DIS
LIN {X 0.008,Y -178.771,Z 1397.441,A 0.000,B 0.000,C 90.000,E1 259.454} C_DIS
LIN {X 0.079,Y -175.818,Z 1397.413,A 0.000,B 0.000,C 90.000,E1 254.338} C_DIS
LIN {X 0.073,Y -172.005,Z 1397.385,A 0.000,B 0.000,C 90.000,E1 249.209} C_DIS
LIN {X 0.047,Y -171.422,Z 1397.380,A 0.000,B 0.000,C 90.000,E1 248.358} C_DIS
LIN {X -0.056,Y -167.660,Z 1397.356,A 0.000,B 0.000,C 90.000,E1 244.076} C_DIS
LIN {X 0.032,Y -166.327,Z 1397.346,A 0.000,B 0.000,C 90.000,E1 242.308} C_DIS
LIN {X 0.018,Y -163.067,Z 1397.327,A 0.000,B 0.000,C 90.000,E1 238.820} C_DIS
LIN {X -0.071,Y -161.005,Z 1397.312,A 0.000,B 0.000,C 90.000,E1 236.215} C_DIS
LIN {X 0.040,Y -157.750,Z 1397.292,A 0.000,B 0.000,C 90.000,E1 232.637} C_DIS
LIN {X -0.023,Y -155.788,Z 1397.278,A 0.000,B 0.000,C 90.000,E1 229.989} C_DIS
LIN {X 0.033,Y -152.041,Z 1397.253,A 0.000,B 0.000,C 90.000,E1 225.486} C_DIS
LIN {X 0.049,Y -150.291,Z 1397.238,A 0.000,B 0.000,C 90.000,E1 222.771} C_DIS
LIN {X -0.024,Y -147.038,Z 1397.213,A 0.000,B 0.000,C 90.000,E1 218.257} C_DIS
LIN {X -0.031,Y -145.618,Z 1397.197,A 0.000,B 0.000,C 90.000,E1 215.518} C_DIS
LIN {X -0.032,Y -143.003,Z 1397.172,A 0.000,B 0.000,C 90.000,E1 210.924} C_DIS
LIN {X 0.025,Y -141.630,Z 1397.151,A 0.000,B 0.000,C 90.000,E1 207.206} C_DIS
LIN {X -0.049,Y -139.435,Z 1397.115,A 0.000,B 0.000,C 90.000,E1 200.737} C_DIS
LIN {X 0.004,Y -139.167,Z 1397.105,A 0.000,B 0.000,C 90.000,E1 198.852} C_DIS
LIN {X 0.038,Y -138.316,Z 1397.053,A 0.000,B 0.000,C 90.000,E1 189.500} C_DIS
LIN {X 0.049,Y -139.476,Z 1397.006,A 0.000,B 0.000,C 90.000,E1 181.088} C_DIS
LIN {X -0.010,Y -141.056,Z 1396.975,A 0.000,B 0.000,C 90.000,E1 175.527} C_DIS
LIN {X -0.056,Y -142.429,Z 1396.960,A 0.000,B 0.000,C 90.000,E1 172.761} C_DIS
LIN {X 0.005,Y -144.666,Z 1396.934,A 0.000,B 0.000,C 90.000,E1 168.117} C_DIS
LIN {X -0.011,Y -147.251,Z 1396.914,A 0.000,B 0.000,C 90.000,E1 164.448} C_DIS
LIN {X 0.006,Y -150.568,Z 1396.888,A 0.000,B 0.000,C 90.000,E1 159.880} C_DIS
LIN {X 0.085,Y -154.037,Z 1396.868,A 0.000,B 0.000,C 90.000,E1 156.230} C_DIS
LIN {X 0.013,Y -157.454,Z 1396.848,A 0.000,B 0.000,C 90.000,E1 152.666} C_DIS
LIN {X -0.039,Y -161.673,Z 1396.828,A 0.000,B 0.000,C 90.000,E1 149.125} C_DIS
LIN {X -0.021,Y -165.868,Z 1396.809,A 0.000,B 0.000,C 90.000,E1 145.595} C_DIS
LIN {X -0.030,Y -170.845,Z 1396.789,A 0.000,B 0.000,C 90.000,E1 142.110} C_DIS
LIN {X 0.017,Y -175.714,Z 1396.770,A 0.000,B 0.000,C 90.000,E1 138.647} C_DIS
LIN {X 0.008,Y -181.326,Z 1396.751,A 0.000,B 0.000,C 90.000,E1 135.243} C_DIS
LIN {X 0.002,Y -186.811,Z 1396.733,A 0.000,B 0.000,C 90.000,E1 131.881} C_DIS
LIN {X -0.052,Y -191.401,Z 1396.719,A 0.000,B 0.000,C 90.000,E1 129.402} C_DIS
LIN {X 0.031,Y -197.247,Z 1396.701,A 0.000,B 0.000,C 90.000,E1 126.091} C_DIS
LIN {X -0.002,Y -199.485,Z 1396.694,A 0.000,B 0.000,C 90.000,E1 124.978} C_DIS
LIN {X -0.052,Y -310.476,Z 1396.694,A 0.000,B 0.000,C 90.000,E1 124.978} C_DIS
LIN {X -0.103,Y -316.577,Z 1396.693,A 0.000,B 0.000,C 90.000,E1 124.739} C_DIS
LIN {X -0.073,Y -319.408,Z 1396.692,A 0.000,B 0.000,C 90.000,E1 124.485} C_DIS
LIN {X -0.140,Y -323.125,Z 1396.689,A 0.000,B 0.000,C 90.000,E1 123.992} C_DIS
LIN {X -0.061,Y -324.764,Z 1396.687,A 0.000,B 0.000,C 90.000,E1 123.658} C_DIS
LIN {X 0.024,Y -327.138,Z 1396.683,A 0.000,B 0.000,C 90.000,E1 123.007} C_DIS
LIN {X -0.123,Y -337.701,Z 1396.668,A 0.000,B 0.000,C 90.000,E1 120.207} C_DIS
LIN {X 0.173,Y -349.611,Z 1396.652,A 0.000,B 0.000,C 90.000,E1 117.385} C_DIS
LIN {X 0.006,Y -362.978,Z 1396.637,A 0.000,B 0.000,C 90.000,E1 114.695} C_DIS
LIN {X -0.011,Y -376.172,Z 1396.624,A 0.000,B 0.000,C 90.000,E1 112.333} C_DIS
LIN {X 0.169,Y -390.697,Z 1396.611,A 0.000,B 0.000,C 90.000,E1 109.993} C_DIS
LIN {X -0.053,Y -406.655,Z 1396.599,A 0.000,B 0.000,C 90.000,E1 107.764} C_DIS
LIN {X -0.002,Y -424.156,Z 1396.586,A 0.000,B 0.000,C 90.000,E1 105.552} C_DIS
LIN {X -0.033,Y -443.298,Z 1396.574,A 0.000,B 0.000,C 90.000,E1 103.411} C_DIS
LIN {X -0.160,Y -463.380,Z 1396.563,A 0.000,B 0.000,C 90.000,E1 101.422} C_DIS
LIN {X 0.038,Y -483.942,Z 1396.553,A 0.000,B 0.000,C 90.000,E1 99.557} C_DIS
LIN {X 0.130,Y -485.975,Z 1396.552,A 0.000,B 0.000,C 90.000,E1 99.321} C_DIS
LIN {X 0.143,Y -487.526,Z 1396.551,A 0.000,B 0.000,C 90.000,E1 99.095} C_DIS
LIN {X 0.039,Y -488.827,Z 1396.549,A 0.000,B 0.000,C 90.000,E1 98.859} C_DIS
LIN {X -0.068,Y -489.783,Z 1396.548,A 0.000,B 0.000,C 90.000,E1 98.624} C_DIS
LIN {X 0.145,Y -490.835,Z 1396.545,A 0.000,B 0.000,C 90.000,E1 98.106} C_DIS
LIN {X -0.120,Y -490.880,Z 1396.542,A 0.000,B 0.000,C 90.000,E1 97.644} C_DIS
LIN {X 0.108,Y -489.924,Z 1396.540,A 0.000,B 0.000,C 90.000,E1 97.125} C_DIS
LIN {X -0.148,Y -487.802,Z 1396.537,A 0.000,B 0.000,C 90.000,E1 96.663} C_DIS
LIN {X -0.127,Y -468.170,Z 1396.520,A 0.000,B 0.000,C 90.000,E1 93.669} C_DIS
LIN {X -0.197,Y -459.933,Z 1396.513,A 0.000,B 0.000,C 90.000,E1 92.407} C_DIS
LIN {X 0.135,Y -440.329,Z 1396.496,A 0.000,B 0.000,C 90.000,E1 89.255} C_DIS
LIN {X 0.126,Y -428.219,Z 1396.484,A 0.000,B 0.000,C 90.000,E1 87.135} C_DIS
LIN {X 0.172,Y -417.538,Z 1396.474,A 0.000,B 0.000,C 90.000,E1 85.241} C_DIS
LIN {X -0.035,Y -408.234,Z 1396.465,A 0.000,B 0.000,C 90.000,E1 83.628} C_DIS
LIN {X 0.135,Y -397.260,Z 1396.454,A 0.000,B 0.000,C 90.000,E1 81.659} C_DIS
LIN {X 0.024,Y -387.728,Z 1396.444,A 0.000,B 0.000,C 90.000,E1 79.982} C_DIS
LIN {X -0.081,Y -374.779,Z 1396.432,A 0.000,B 0.000,C 90.000,E1 77.701} C_DIS
LIN {X -0.005,Y -365.041,Z 1396.422,A 0.000,B 0.000,C 90.000,E1 75.936} C_DIS
LIN {X -0.019,Y -355.147,Z 1396.412,A 0.000,B 0.000,C 90.000,E1 74.157} C_DIS
LIN {X -0.114,Y -345.196,Z 1396.402,A 0.000,B 0.000,C 90.000,E1 72.362} C_DIS
LIN {X 0.030,Y -333.490,Z 1396.390,A 0.000,B 0.000,C 90.000,E1 70.188} C_DIS
LIN {X -0.017,Y -317.146,Z 1396.372,A 0.000,B 0.000,C 90.000,E1 67.050} C_DIS
LIN {X -0.045,Y -302.154,Z 1396.354,A 0.000,B 0.000,C 90.000,E1 63.819} C_DIS
LIN {X -0.091,Y -291.496,Z 1396.340,A 0.000,B 0.000,C 90.000,E1 61.179} C_DIS
LIN {X 0.022,Y -281.830,Z 1396.325,A 0.000,B 0.000,C 90.000,E1 58.456} C_DIS
LIN {X -0.004,Y -270.918,Z 1396.306,A 0.000,B 0.000,C 90.000,E1 55.022} C_DIS
LIN {X -0.099,Y -260.734,Z 1396.286,A 0.000,B 0.000,C 90.000,E1 51.537} C_DIS
LIN {X 0.095,Y -251.134,Z 1396.266,A 0.000,B 0.000,C 90.000,E1 47.919} C_DIS
LIN {X 0.119,Y -242.279,Z 1396.246,A 0.000,B 0.000,C 90.000,E1 44.271} C_DIS
LIN {X -0.111,Y -234.263,Z 1396.225,A 0.000,B 0.000,C 90.000,E1 40.620} C_DIS
LIN {X 0.013,Y -227.147,Z 1396.205,A 0.000,B 0.000,C 90.000,E1 36.824} C_DIS
LIN {X 0.001,Y -220.892,Z 1396.183,A 0.000,B 0.000,C 90.000,E1 33.007} C_DIS
LIN {X -0.061,Y -215.576,Z 1396.162,A 0.000,B 0.000,C 90.000,E1 29.155} C_DIS
LIN {X 0.074,Y -211.151,Z 1396.140,A 0.000,B 0.000,C 90.000,E1 25.207} C_DIS
LIN {X 0.018,Y -207.117,Z 1396.114,A 0.000,B 0.000,C 90.000,E1 20.482} C_DIS
LIN {X -0.029,Y -204.222,Z 1396.087,A 0.000,B 0.000,C 90.000,E1 15.717} C_DIS
LIN {X -0.032,Y -202.306,Z 1396.065,A 0.000,B 0.000,C 90.000,E1 11.715} C_DIS
LIN {X -0.071,Y -200.976,Z 1396.047,A 0.000,B 0.000,C 90.000,E1 8.511} C_DIS
LIN {X -0.049,Y -199.577,Z 1396.025,A 0.000,B 0.000,C 90.000,E1 4.473} C_DIS
LIN {X 0.078,Y -198.672,Z 1396.007,A 0.000,B 0.000,C 90.000,E1 1.203} C_DIS
LIN {X 0.050,Y -197.718,Z 1395.979,A 0.000,B 0.000,C 90.000,E1 356.274} C_DIS
LIN {X -0.058,Y -197.568,Z 1395.948,A 0.000,B 0.000,C 90.000,E1 350.622} C_DIS
LIN {X 0.027,Y -199.776,Z 1395.903,A 0.000,B 0.000,C 90.000,E1 342.489} C_DIS
LIN {X -0.037,Y -202.811,Z 1395.876,A 0.000,B 0.000,C 90.000,E1 337.667} C_DIS
LIN {X 0.036,Y -206.607,Z 1395.854,A 0.000,B 0.000,C 90.000,E1 333.640} C_DIS
LIN {X 0.049,Y -211.463,Z 1395.832,A 0.000,B 0.000,C 90.000,E1 329.665} C_DIS
LIN {X -0.014,Y -217.620,Z 1395.810,A 0.000,B 0.000,C 90.000,E1 325.754} C_DIS
LIN {X 0.032,Y -223.549,Z 1395.792,A 0.000,B 0.000,C 90.000,E1 322.637} C_DIS
LIN {X -0.020,Y -230.423,Z 1395.775,A 0.000,B 0.000,C 90.000,E1 319.585} C_DIS
LIN {X -0.124,Y -239.144,Z 1395.757,A 0.000,B 0.000,C 90.000,E1 316.215} C_DIS
LIN {X 0.026,Y -248.928,Z 1395.738,A 0.000,B 0.000,C 90.000,E1 312.852} C_DIS
LIN {X 0.118,Y -258.865,Z 1395.722,A 0.000,B 0.000,C 90.000,E1 309.930} C_DIS
LIN {X 0.082,Y -271.415,Z 1395.704,A 0.000,B 0.000,C 90.000,E1 306.744} C_DIS
LIN {X -0.085,Y -280.651,Z 1395.693,A 0.000,B 0.000,C 90.000,E1 304.692} C_DIS
LIN {X 0.015,Y -289.270,Z 1395.683,A 0.000,B 0.000,C 90.000,E1 302.959} C_DIS
LIN {X 0.104,Y -296.986,Z 1395.676,A 0.000,B 0.000,C 90.000,E1 301.592} C_DIS
LIN {X 0.038,Y -310.095,Z 1395.665,A 0.000,B 0.000,C 90.000,E1 299.617} C_DIS
LIN {X -0.094,Y -317.231,Z 1395.659,A 0.000,B 0.000,C 90.000,E1 298.693} C_DIS
LIN {X -0.065,Y -329.958,Z 1395.651,A 0.000,B 0.000,C 90.000,E1 297.180} C_DIS
LIN {X -0.108,Y -346.259,Z 1395.641,A 0.000,B 0.000,C 90.000,E1 295.412} C_DIS
LIN {X -0.131,Y -362.281,Z 1395.631,A 0.000,B 0.000,C 90.000,E1 293.695} C_DIS
LIN {X 0.180,Y -372.688,Z 1395.625,A 0.000,B 0.000,C 90.000,E1 292.514} C_DIS
LIN {X -0.031,Y -382.890,Z 1395.619,A 0.000,B 0.000,C 90.000,E1 291.408} C_DIS
LIN {X -0.022,Y -395.244,Z 1395.611,A 0.000,B 0.000,C 90.000,E1 289.993} C_DIS
LIN {X -0.007,Y -415.199,Z 1395.599,A 0.000,B 0.000,C 90.000,E1 287.764} C_DIS
LIN {X 0.250,Y -422.478,Z 1395.594,A 0.000,B 0.000,C 90.000,E1 286.913} C_DIS
LIN {X -0.007,Y -429.273,Z 1395.590,A 0.000,B 0.000,C 90.000,E1 286.134} C_DIS
LIN {X -0.090,Y -433.402,Z 1395.587,A 0.000,B 0.000,C 90.000,E1 285.607} C_DIS
LIN {X 0.158,Y -438.923,Z 1395.582,A 0.000,B 0.000,C 90.000,E1 284.773} C_DIS
LIN {X -0.073,Y -443.598,Z 1395.578,A 0.000,B 0.000,C 90.000,E1 284.008} C_DIS
LIN {X -0.164,Y -447.392,Z 1395.573,A 0.000,B 0.000,C 90.000,E1 283.231} C_DIS
LIN {X -0.130,Y -449.505,Z 1395.570,A 0.000,B 0.000,C 90.000,E1 282.703} C_DIS
LIN {X -0.083,Y -451.263,Z 1395.568,A 0.000,B 0.000,C 90.000,E1 282.175} C_DIS
LIN {X -0.120,Y -452.712,Z 1395.565,A 0.000,B 0.000,C 90.000,E1 281.658} C_DIS
LIN {X -0.053,Y -453.779,Z 1395.562,A 0.000,B 0.000,C 90.000,E1 281.130} C_DIS
LIN {X 0.021,Y -454.427,Z 1395.559,A 0.000,B 0.000,C 90.000,E1 280.602} C_DIS
LIN {X 0.098,Y -454.711,Z 1395.556,A 0.000,B 0.000,C 90.000,E1 280.074} C_DIS
LIN {X 0.101,Y -454.539,Z 1395.553,A 0.000,B 0.000,C 90.000,E1 279.557} C_DIS
LIN {X 0.180,Y -453.848,Z 1395.550,A 0.000,B 0.000,C 90.000,E1 279.029} C_DIS
LIN {X 0.187,Y -452.722,Z 1395.547,A 0.000,B 0.000,C 90.000,E1 278.511} C_DIS
LIN {X 0.192,Y -451.012,Z 1395.545,A 0.000,B 0.000,C 90.000,E1 277.992} C_DIS
LIN {X 0.192,Y -448.651,Z 1395.542,A 0.000,B 0.000,C 90.000,E1 277.473} C_DIS
LIN {X -0.009,Y -447.239,Z 1395.540,A 0.000,B 0.000,C 90.000,E1 277.239} C_DIS
LIN {X -0.032,Y -443.734,Z 1395.537,A 0.000,B 0.000,C 90.000,E1 276.720} C_DIS
LIN {X -0.071,Y -439.274,Z 1395.534,A 0.000,B 0.000,C 90.000,E1 276.201} C_DIS
LIN {X -0.043,Y -433.799,Z 1395.531,A 0.000,B 0.000,C 90.000,E1 275.682} C_DIS
LIN {X -0.133,Y -427.667,Z 1395.529,A 0.000,B 0.000,C 90.000,E1 275.220} C_DIS
LIN {X 0.200,Y -421.313,Z 1395.527,A 0.000,B 0.000,C 90.000,E1 274.759} C_DIS
LIN {X 0.055,Y -414.661,Z 1395.525,A 0.000,B 0.000,C 90.000,E1 274.416} C_DIS
LIN {X -0.145,Y -408.168,Z 1395.523,A 0.000,B 0.000,C 90.000,E1 274.131} C_DIS
LIN {X 0.170,Y -398.351,Z 1395.521,A 0.000,B 0.000,C 90.000,E1 273.669} C_DIS
LIN {X -0.004,Y -388.641,Z 1395.518,A 0.000,B 0.000,C 90.000,E1 273.326} C_DIS
LIN {X 0.053,Y -378.605,Z 1395.517,A 0.000,B 0.000,C 90.000,E1 272.980} C_DIS
LIN {X 0.047,Y -367.980,Z 1395.515,A 0.000,B 0.000,C 90.000,E1 272.694} C_DIS
LIN {X 0.071,Y -357.399,Z 1395.514,A 0.000,B 0.000,C 90.000,E1 272.465} C_DIS
LIN {X -0.005,Y -344.729,Z 1395.513,A 0.000,B 0.000,C 90.000,E1 272.293} C_DIS
LIN {X 0.007,Y -331.484,Z 1395.512,A 0.000,B 0.000,C 90.000,E1 272.178} C_DIS
LIN {X 0.069,Y -319.095,Z 1395.512,A 0.000,B 0.000,C 90.000,E1 272.121} C_DIS
LIN {X 0.012,Y -181.242,Z 1395.512,A 0.000,B 0.000,C 90.000,E1 272.121} C_DIS
LIN {X 0.017,Y -181.576,Z 1395.502,A 0.000,B 0.000,C 90.000,E1 270.401} C_DIS
LIN {X -0.007,Y -180.906,Z 1395.474,A 0.000,B 0.000,C 90.000,E1 265.355} C_DIS
LIN {X 0.067,Y -180.681,Z 1395.469,A 0.000,B 0.000,C 90.000,E1 264.489} C_DIS
LIN {X -0.034,Y -178.764,Z 1395.441,A 0.000,B 0.000,C 90.000,E1 259.454} C_DIS
LIN {X 0.038,Y -175.811,Z 1395.413,A 0.000,B 0.000,C 90.000,E1 254.338} C_DIS
LIN {X 0.031,Y -171.997,Z 1395.385,A 0.000,B 0.000,C 90.000,E1 249.209} C_DIS
LIN {X 0.007,Y -171.410,Z 1395.380,A 0.000,B 0.000,C 90.000,E1 248.358} C_DIS
LIN {X 0.054,Y -167.649,Z 1395.356,A 0.000,B 0.000,C 90.000,E1 244.024} C_DIS
LIN {X 0.069,Y -166.313,Z 1395.346,A 0.000,B 0.000,C 90.000,E1 242.281} C_DIS
LIN {X 0.062,Y -163.055,Z 1395.327,A 0.000,B 0.000,C 90.000,E1 238.791} C_DIS
LIN {X 0.023,Y -160.991,Z 1395.312,A 0.000,B 0.000,C 90.000,E1 236.167} C_DIS
LIN {X 0.001,Y -157.739,Z 1395.292,A 0.000,B 0.000,C 90.000,E1 232.637} C_DIS
LIN {X -0.061,Y -155.777,Z 1395.278,A 0.000,B 0.000,C 90.000,E1 229.989} C_DIS
LIN {X -0.005,Y -152.031,Z 1395.253,A 0.000,B 0.000,C 90.000,E1 225.486} C_DIS
LIN {X 0.012,Y -150.279,Z 1395.238,A 0.000,B 0.000,C 90.000,E1 222.771} C_DIS
LIN {X -0.062,Y -147.030,Z 1395.212,A 0.000,B 0.000,C 90.000,E1 218.257} C_DIS
LIN {X -0.068,Y -145.611,Z 1395.197,A 0.000,B 0.000,C 90.000,E1 215.518} C_DIS
LIN {X 0.054,Y -142.996,Z 1395.172,A 0.000,B 0.000,C 90.000,E1 210.875} C_DIS
LIN {X -0.011,Y -141.623,Z 1395.151,A 0.000,B 0.000,C 90.000,E1 207.206} C_DIS
LIN {X -0.086,Y -139.432,Z 1395.115,A 0.000,B 0.000,C 90.000,E1 200.737} C_DIS
LIN {X -0.031,Y -139.163,Z 1395.105,A 0.000,B 0.000,C 90.000,E1 198.852} C_DIS
LIN {X 0.006,Y -138.340,Z 1395.058,A 0.000,B 0.000,C 90.000,E1 190.433} C_DIS
LIN {X 0.013,Y -139.477,Z 1395.006,A 0.000,B 0.000,C 90.000,E1 181.088} C_DIS
LIN {X -0.047,Y -141.063,Z 1394.975,A 0.000,B 0.000,C 90.000,E1 175.527} C_DIS
LIN {X 0.048,Y -142.437,Z 1394.960,A 0.000,B 0.000,C 90.000,E1 172.704} C_DIS
LIN {X -0.032,Y -144.675,Z 1394.934,A 0.000,B 0.000,C 90.000,E1 168.117} C_DIS
LIN {X -0.049,Y -147.263,Z 1394.913,A 0.000,B 0.000,C 90.000,E1 164.448} C_DIS
LIN {X -0.032,Y -150.580,Z 1394.888,A 0.000,B 0.000,C 90.000,E1 159.880} C_DIS
LIN {X 0.047,Y -154.052,Z 1394.868,A 0.000,B 0.000,C 90.000,E1 156.230} C_DIS
LIN {X -0.026,Y -157.469,Z 1394.848,A 0.000,B 0.000,C 90.000,E1 152.666} C_DIS
LIN {X 0.061,Y -161.691,Z 1394.828,A 0.000,B 0.000,C 90.000,E1 149.076} C_DIS
LIN {X -0.061,Y -165.885,Z 1394.809,A 0.000,B 0.000,C 90.000,E1 145.595} C_DIS
LIN {X -0.072,Y -170.866,Z 1394.789,A 0.000,B 0.000,C 90.000,E1 142.110} C_DIS
LIN {X -0.025,Y -175.735,Z 1394.770,A 0.000,B 0.000,C 90.000,E1 138.647} C_DIS
LIN {X -0.036,Y -181.346,Z 1394.751,A 0.000,B 0.000,C 90.000,E1 135.243} C_DIS
LIN {X 0.099,Y -186.835,Z 1394.733,A 0.000,B 0.000,C 90.000,E1 131.838} C_DIS
LIN {X 0.053,Y -191.422,Z 1394.719,A 0.000,B 0.000,C 90.000,E1 129.358} C_DIS
LIN {X -0.015,Y -197.272,Z 1394.700,A 0.000,B 0.000,C 90.000,E1 126.091} C_DIS
LIN {X -0.097,Y -199.445,Z 1394.694,A 0.000,B 0.000,C 90.000,E1 125.025} C_DIS
LIN {X 0.067,Y -309.547,Z 1394.694,A 0.000,B 0.000,C 90.000,E1 124.978} C_DIS
LIN {X 0.058,Y -311.879,Z 1394.694,A 0.000,B 0.000,C 90.000,E1 124.945} C_DIS
LIN {X 0.087,Y -316.885,Z 1394.693,A 0.000,B 0.000,C 90.000,E1 124.692} C_DIS
LIN {X 0.035,Y -319.597,Z 1394.691,A 0.000,B 0.000,C 90.000,E1 124.452} C_DIS
LIN {X 0.135,Y -323.314,Z 1394.688,A 0.000,B 0.000,C 90.000,E1 123.913} C_DIS
LIN {X -0.055,Y -324.894,Z 1394.687,A 0.000,B 0.000,C 90.000,E1 123.627} C_DIS
LIN {X -0.005,Y -331.763,Z 1394.676,A 0.000,B 0.000,C 90.000,E1 121.720} C_DIS
LIN {X -0.191,Y -342.928,Z 1394.661,A 0.000,B 0.000,C 90.000,E1 118.949} C_DIS
LIN {X -0.070,Y -355.486,Z 1394.645,A 0.000,B 0.000,C 90.000,E1 116.181} C_DIS
LIN {X 0.109,Y -369.552,Z 1394.630,A 0.000,B 0.000,C 90.000,E1 113.462} C_DIS
LIN {X -0.085,Y -383.416,Z 1394.617,A 0.000,B 0.000,C 90.000,E1 111.153} C_DIS
LIN {X 0.006,Y -398.661,Z 1394.605,A 0.000,B 0.000,C 90.000,E1 108.852} C_DIS
LIN {X -0.019,Y -415.395,Z 1394.592,A 0.000,B 0.000,C 90.000,E1 106.622} C_DIS
LIN {X 0.138,Y -433.734,Z 1394.580,A 0.000,B 0.000,C 90.000,E1 104.426} C_DIS
LIN {X 0.029,Y -453.488,Z 1394.569,A 0.000,B 0.000,C 90.000,E1 102.355} C_DIS
LIN {X 0.054,Y -473.856,Z 1394.558,A 0.000,B 0.000,C 90.000,E1 100.433} C_DIS
LIN {X -0.148,Y -484.121,Z 1394.553,A 0.000,B 0.000,C 90.000,E1 99.557} C_DIS
LIN {X -0.082,Y -486.092,Z 1394.552,A 0.000,B 0.000,C 90.000,E1 99.321} C_DIS
LIN {X -0.092,Y -487.597,Z 1394.550,A 0.000,B 0.000,C 90.000,E1 99.095} C_DIS
LIN {X -0.197,Y -488.840,Z 1394.549,A 0.000,B 0.000,C 90.000,E1 98.859} C_DIS
LIN {X 0.180,Y -489.748,Z 1394.548,A 0.000,B 0.000,C 90.000,E1 98.568} C_DIS
LIN {X -0.091,Y -490.720,Z 1394.545,A 0.000,B 0.000,C 90.000,E1 98.106} C_DIS
LIN {X 0.130,Y -490.689,Z 1394.542,A 0.000,B 0.000,C 90.000,E1 97.587} C_DIS
LIN {X -0.129,Y -489.653,Z 1394.540,A 0.000,B 0.000,C 90.000,E1 97.125} C_DIS
LIN {X -0.228,Y -488.712,Z 1394.538,A 0.000,B 0.000,C 90.000,E1 96.891} C_DIS
LIN {X 0.099,Y -487.428,Z 1394.537,A 0.000,B 0.000,C 90.000,E1 96.606} C_DIS
LIN {X 0.095,Y -467.742,Z 1394.520,A 0.000,B 0.000,C 90.000,E1 93.612} C_DIS
LIN {X 0.015,Y -459.464,Z 1394.513,A 0.000,B 0.000,C 90.000,E1 92.350} C_DIS
LIN {X -0.116,Y -439.940,Z 1394.496,A 0.000,B 0.000,C 90.000,E1 89.255} C_DIS
LIN {X -0.129,Y -427.859,Z 1394.484,A 0.000,B 0.000,C 90.000,E1 87.135} C_DIS
LIN {X -0.187,Y -418.743,Z 1394.475,A 0.000,B 0.000,C 90.000,E1 85.527} C_DIS
LIN {X 0.116,Y -407.906,Z 1394.464,A 0.000,B 0.000,C 90.000,E1 83.571} C_DIS
LIN {X 0.194,Y -398.577,Z 1394.455,A 0.000,B 0.000,C 90.000,E1 81.894} C_DIS
LIN {X 0.153,Y -387.459,Z 1394.444,A 0.000,B 0.000,C 90.000,E1 79.926} C_DIS
LIN {X 0.034,Y -374.508,Z 1394.431,A 0.000,B 0.000,C 90.000,E1 77.645} C_DIS
LIN {X 0.100,Y -364.764,Z 1394.422,A 0.000,B 0.000,C 90.000,E1 75.880} C_DIS
LIN {X 0.075,Y -354.856,Z 1394.412,A 0.000,B 0.000,C 90.000,E1 74.102} C_DIS
LIN {X -0.030,Y -344.892,Z 1394.402,A 0.000,B 0.000,C 90.000,E1 72.308} C_DIS
LIN {X 0.100,Y -333.182,Z 1394.390,A 0.000,B 0.000,C 90.000,E1 70.134} C_DIS
LIN {X 0.090,Y -318.428,Z 1394.374,A 0.000,B 0.000,C 90.000,E1 67.305} C_DIS
LIN {X -0.011,Y -301.912,Z 1394.354,A 0.000,B 0.000,C 90.000,E1 63.768} C_DIS
LIN {X -0.071,Y -291.279,Z 1394.339,A 0.000,B 0.000,C 90.000,E1 61.129} C_DIS
LIN {X 0.029,Y -281.649,Z 1394.324,A 0.000,B 0.000,C 90.000,E1 58.408} C_DIS
LIN {X -0.011,Y -270.785,Z 1394.305,A 0.000,B 0.000,C 90.000,E1 54.975} C_DIS
LIN {X 0.043,Y -260.634,Z 1394.286,A 0.000,B 0.000,C 90.000,E1 51.457} C_DIS
LIN {X 0.063,Y -251.093,Z 1394.266,A 0.000,B 0.000,C 90.000,E1 47.877} C_DIS
LIN {X -0.094,Y -242.266,Z 1394.246,A 0.000,B 0.000,C 90.000,E1 44.271} C_DIS
LIN {X 0.015,Y -234.272,Z 1394.225,A 0.000,B 0.000,C 90.000,E1 40.539} C_DIS
LIN {X -0.049,Y -227.179,Z 1394.204,A 0.000,B 0.000,C 90.000,E1 36.790} C_DIS
LIN {X -0.005,Y -220.972,Z 1394.183,A 0.000,B 0.000,C 90.000,E1 32.959} C_DIS
LIN {X 0.048,Y -215.695,Z 1394.162,A 0.000,B 0.000,C 90.000,E1 29.077} C_DIS
LIN {X 0.088,Y -211.314,Z 1394.140,A 0.000,B 0.000,C 90.000,E1 25.155} C_DIS
LIN {X 0.046,Y -207.352,Z 1394.114,A 0.000,B 0.000,C 90.000,E1 20.429} C_DIS
LIN {X 0.013,Y -204.511,Z 1394.087,A 0.000,B 0.000,C 90.000,E1 15.662} C_DIS
LIN {X 0.022,Y -202.594,Z 1394.065,A 0.000,B 0.000,C 90.000,E1 11.658} C_DIS
LIN {X 0.011,Y -200.934,Z 1394.042,A 0.000,B 0.000,C 90.000,E1 7.644} C_DIS
LIN {X 0.012,Y -199.607,Z 1394.020,A 0.000,B 0.000,C 90.000,E1 3.612} C_DIS
LIN {X -0.036,Y -198.524,Z 1393.997,A 0.000,B 0.000,C 90.000,E1 359.542} C_DIS
LIN {X 0.008,Y -197.766,Z 1393.970,A 0.000,B 0.000,C 90.000,E1 354.666} C_DIS
LIN {X -0.021,Y -197.955,Z 1393.939,A 0.000,B 0.000,C 90.000,E1 348.993} C_DIS
LIN {X 0.018,Y -200.406,Z 1393.898,A 0.000,B 0.000,C 90.000,E1 341.692} C_DIS
LIN {X -0.018,Y -203.696,Z 1393.871,A 0.000,B 0.000,C 90.000,E1 336.869} C_DIS
LIN {X -0.020,Y -207.689,Z 1393.849,A 0.000,B 0.000,C 90.000,E1 332.871} C_DIS
LIN {X -0.053,Y -212.799,Z 1393.827,A 0.000,B 0.000,C 90.000,E1 328.918} C_DIS
LIN {X 0.048,Y -219.225,Z 1393.806,A 0.000,B 0.000,C 90.000,E1 324.975} C_DIS
LIN {X -0.041,Y -225.373,Z 1393.788,A 0.000,B 0.000,C 90.000,E1 321.904} C_DIS
LIN {X -0.048,Y -232.454,Z 1393.771,A 0.000,B 0.000,C 90.000,E1 318.852} C_DIS
LIN {X -0.104,Y -241.389,Z 1393.753,A 0.000,B 0.000,C 90.000,E1 315.486} C_DIS
LIN {X -0.060,Y -250.245,Z 1393.736,A 0.000,B 0.000,C 90.000,E1 312.528} C_DIS
LIN {X -0.109,Y -260.291,Z 1393.720,A 0.000,B 0.000,C 90.000,E1 309.644} C_DIS
LIN {X 0.048,Y -272.992,Z 1393.702,A 0.000,B 0.000,C 90.000,E1 306.423} C_DIS
LIN {X 0.132,Y -282.380,Z 1393.691,A 0.000,B 0.000,C 90.000,E1 304.326} C_DIS
LIN {X 0.111,Y -291.180,Z 1393.681,A 0.000,B 0.000,C 90.000,E1 302.625} C_DIS
LIN {X -0.182,Y -299.112,Z 1393.674,A 0.000,B 0.000,C 90.000,E1 301.337} C_DIS
LIN {X -0.102,Y -310.126,Z 1393.665,A 0.000,B 0.000,C 90.000,E1 299.667} C_DIS
LIN {X -0.053,Y -320.077,Z 1393.657,A 0.000,B 0.000,C 90.000,E1 298.359} C_DIS
LIN {X -0.114,Y -335.997,Z 1393.647,A 0.000,B 0.000,C 90.000,E1 296.539} C_DIS
LIN {X -0.056,Y -349.420,Z 1393.639,A 0.000,B 0.000,C 90.000,E1 295.079} C_DIS
LIN {X -0.070,Y -362.812,Z 1393.631,A 0.000,B 0.000,C 90.000,E1 293.643} C_DIS
LIN {X -0.131,Y -373.260,Z 1393.625,A 0.000,B 0.000,C 90.000,E1 292.514} C_DIS
LIN {X -0.058,Y -383.516,Z 1393.619,A 0.000,B 0.000,C 90.000,E1 291.354} C_DIS
LIN {X -0.102,Y -395.917,Z 1393.611,A 0.000,B 0.000,C 90.000,E1 289.939} C_DIS
LIN {X 0.038,Y -415.882,Z 1393.598,A 0.000,B 0.000,C 90.000,E1 287.692} C_DIS
LIN {X 0.139,Y -423.156,Z 1393.594,A 0.000,B 0.000,C 90.000,E1 286.858} C_DIS
LIN {X -0.023,Y -429.823,Z 1393.589,A 0.000,B 0.000,C 90.000,E1 286.079} C_DIS
LIN {X 0.191,Y -435.815,Z 1393.585,A 0.000,B 0.000,C 90.000,E1 285.245} C_DIS
LIN {X 0.153,Y -439.400,Z 1393.582,A 0.000,B 0.000,C 90.000,E1 284.717} C_DIS
LIN {X 0.036,Y -444.028,Z 1393.578,A 0.000,B 0.000,C 90.000,E1 283.939} C_DIS
LIN {X -0.158,Y -447.801,Z 1393.573,A 0.000,B 0.000,C 90.000,E1 283.175} C_DIS
LIN {X -0.121,Y -449.872,Z 1393.570,A 0.000,B 0.000,C 90.000,E1 282.647} C_DIS
LIN {X -0.070,Y -451.634,Z 1393.567,A 0.000,B 0.000,C 90.000,E1 282.119} C_DIS
LIN {X -0.013,Y -453.036,Z 1393.564,A 0.000,B 0.000,C 90.000,E1 281.591} C_DIS
LIN {X -0.035,Y -454.074,Z 1393.562,A 0.000,B 0.000,C 90.000,E1 281.074} C_DIS
LIN {X 0.042,Y -454.696,Z 1393.559,A 0.000,B 0.000,C 90.000,E1 280.546} C_DIS
LIN {X 0.122,Y -454.923,Z 1393.556,A 0.000,B 0.000,C 90.000,E1 280.018} C_DIS
LIN {X 0.127,Y -454.703,Z 1393.553,A 0.000,B 0.000,C 90.000,E1 279.500} C_DIS
LIN {X 0.209,Y -454.012,Z 1393.550,A 0.000,B 0.000,C 90.000,E1 278.973} C_DIS
LIN {X 0.216,Y -452.819,Z 1393.547,A 0.000,B 0.000,C 90.000,E1 278.454} C_DIS
LIN {X -0.224,Y -451.074,Z 1393.544,A 0.000,B 0.000,C 90.000,E1 277.992} C_DIS
LIN {X -0.162,Y -448.701,Z 1393.541,A 0.000,B 0.000,C 90.000,E1 277.466} C_DIS
LIN {X -0.178,Y -445.601,Z 1393.538,A 0.000,B 0.000,C 90.000,E1 276.947} C_DIS
LIN {X 0.000,Y -443.748,Z 1393.537,A 0.000,B 0.000,C 90.000,E1 276.663} C_DIS
LIN {X -0.038,Y -439.262,Z 1393.534,A 0.000,B 0.000,C 90.000,E1 276.144} C_DIS
LIN {X -0.002,Y -433.743,Z 1393.531,A 0.000,B 0.000,C 90.000,E1 275.625} C_DIS
LIN {X -0.071,Y -427.629,Z 1393.529,A 0.000,B 0.000,C 90.000,E1 275.163} C_DIS
LIN {X -0.133,Y -421.266,Z 1393.526,A 0.000,B 0.000,C 90.000,E1 274.759} C_DIS
LIN {X 0.142,Y -414.620,Z 1393.524,A 0.000,B 0.000,C 90.000,E1 274.359} C_DIS
LIN {X 0.107,Y -404.675,Z 1393.522,A 0.000,B 0.000,C 90.000,E1 273.898} C_DIS
LIN {X 0.142,Y -394.926,Z 1393.520,A 0.000,B 0.000,C 90.000,E1 273.498} C_DIS
LIN {X 0.057,Y -385.032,Z 1393.518,A 0.000,B 0.000,C 90.000,E1 273.154} C_DIS
LIN {X 0.176,Y -378.521,Z 1393.516,A 0.000,B 0.000,C 90.000,E1 272.922} C_DIS
LIN {X 0.163,Y -367.715,Z 1393.515,A 0.000,B 0.000,C 90.000,E1 272.636} C_DIS
LIN {X -0.144,Y -357.103,Z 1393.514,A 0.000,B 0.000,C 90.000,E1 272.465} C_DIS
LIN {X 0.084,Y -347.906,Z 1393.513,A 0.000,B 0.000,C 90.000,E1 272.293} C_DIS
LIN {X -0.060,Y -332.317,Z 1393.512,A 0.000,B 0.000,C 90.000,E1 272.178} C_DIS
LIN {X -0.005,Y -319.162,Z 1393.512,A 0.000,B 0.000,C 90.000,E1 272.121} C_DIS
LIN {X -0.027,Y -181.244,Z 1393.512,A 0.000,B 0.000,C 90.000,E1 272.121} C_DIS
LIN {X -0.066,Y -181.577,Z 1393.502,A 0.000,B 0.000,C 90.000,E1 270.401} C_DIS
LIN {X -0.089,Y -180.905,Z 1393.474,A 0.000,B 0.000,C 90.000,E1 265.355} C_DIS
LIN {X -0.015,Y -180.667,Z 1393.469,A 0.000,B 0.000,C 90.000,E1 264.489} C_DIS
LIN {X 0.059,Y -178.749,Z 1393.441,A 0.000,B 0.000,C 90.000,E1 259.398} C_DIS
LIN {X -0.043,Y -175.796,Z 1393.413,A 0.000,B 0.000,C 90.000,E1 254.338} C_DIS
LIN {X -0.049,Y -171.980,Z 1393.384,A 0.000,B 0.000,C 90.000,E1 249.209} C_DIS
LIN {X -0.010,Y -171.386,Z 1393.380,A 0.000,B 0.000,C 90.000,E1 248.337} C_DIS
LIN {X -0.025,Y -167.630,Z 1393.356,A 0.000,B 0.000,C 90.000,E1 244.024} C_DIS
LIN {X -0.010,Y -166.285,Z 1393.346,A 0.000,B 0.000,C 90.000,E1 242.281} C_DIS
LIN {X -0.015,Y -163.033,Z 1393.327,A 0.000,B 0.000,C 90.000,E1 238.791} C_DIS
LIN {X 0.036,Y -160.962,Z 1393.312,A 0.000,B 0.000,C 90.000,E1 236.135} C_DIS
LIN {X -0.075,Y -157.716,Z 1393.292,A 0.000,B 0.000,C 90.000,E1 232.637} C_DIS
LIN {X 0.083,Y -155.756,Z 1393.277,A 0.000,B 0.000,C 90.000,E1 229.908} C_DIS
LIN {X -0.079,Y -152.012,Z 1393.253,A 0.000,B 0.000,C 90.000,E1 225.486} C_DIS
LIN {X -0.062,Y -150.258,Z 1393.237,A 0.000,B 0.000,C 90.000,E1 222.771} C_DIS
LIN {X 0.072,Y -147.013,Z 1393.212,A 0.000,B 0.000,C 90.000,E1 218.177} C_DIS
LIN {X -0.022,Y -145.596,Z 1393.197,A 0.000,B 0.000,C 90.000,E1 215.471} C_DIS
LIN {X -0.018,Y -142.983,Z 1393.172,A 0.000,B 0.000,C 90.000,E1 210.875} C_DIS
LIN {X -0.018,Y -141.610,Z 1393.151,A 0.000,B 0.000,C 90.000,E1 207.180} C_DIS
LIN {X 0.023,Y -139.426,Z 1393.115,A 0.000,B 0.000,C 90.000,E1 200.663} C_DIS
LIN {X 0.075,Y -139.157,Z 1393.104,A 0.000,B 0.000,C 90.000,E1 198.779} C_DIS
LIN {X -0.040,Y -138.343,Z 1393.058,A 0.000,B 0.000,C 90.000,E1 190.423} C_DIS
LIN {X -0.058,Y -139.482,Z 1393.006,A 0.000,B 0.000,C 90.000,E1 181.088} C_DIS
LIN {X 0.023,Y -141.075,Z 1392.975,A 0.000,B 0.000,C 90.000,E1 175.469} C_DIS
LIN {X -0.024,Y -142.451,Z 1392.959,A 0.000,B 0.000,C 90.000,E1 172.704} C_DIS
LIN {X 0.067,Y -144.692,Z 1392.934,A 0.000,B 0.000,C 90.000,E1 168.049} C_DIS
LIN {X 0.020,Y -147.285,Z 1392.913,A 0.000,B 0.000,C 90.000,E1 164.393} C_DIS
LIN {X 0.035,Y -150.604,Z 1392.888,A 0.000,B 0.000,C 90.000,E1 159.826} C_DIS
LIN {X -0.028,Y -154.078,Z 1392.868,A 0.000,B 0.000,C 90.000,E1 156.230} C_DIS
LIN {X 0.037,Y -157.499,Z 1392.848,A 0.000,B 0.000,C 90.000,E1 152.615} C_DIS
LIN {X -0.018,Y -161.727,Z 1392.828,A 0.000,B 0.000,C 90.000,E1 149.076} C_DIS
LIN {X -0.005,Y -165.921,Z 1392.809,A 0.000,B 0.000,C 90.000,E1 145.548} C_DIS
LIN {X -0.018,Y -170.908,Z 1392.789,A 0.000,B 0.000,C 90.000,E1 142.065} C_DIS
LIN {X 0.009,Y -175.776,Z 1392.770,A 0.000,B 0.000,C 90.000,E1 138.609} C_DIS
LIN {X 0.010,Y -181.385,Z 1392.751,A 0.000,B 0.000,C 90.000,E1 135.202} C_DIS
LIN {X 0.014,Y -186.882,Z 1392.732,A 0.000,B 0.000,C 90.000,E1 131.838} C_DIS
LIN {X -0.034,Y -191.465,Z 1392.719,A 0.000,B 0.000,C 90.000,E1 129.358} C_DIS
LIN {X -0.102,Y -197.321,Z 1392.700,A 0.000,B 0.000,C 90.000,E1 126.091} C_DIS
LIN {X -0.054,Y -199.419,Z 1392.694,A 0.000,B 0.000,C 90.000,E1 125.025} C_DIS
LIN {X -0.133,Y -309.973,Z 1392.694,A 0.000,B 0.000,C 90.000,E1 125.025} C_DIS
LIN {X 0.185,Y -314.779,Z 1392.694,A 0.000,B 0.000,C 90.000,E1 124.818} C_DIS
LIN {X 0.116,Y -316.927,Z 1392.693,A 0.000,B 0.000,C 90.000,E1 124.692} C_DIS
LIN {X 0.159,Y -319.877,Z 1392.691,A 0.000,B 0.000,C 90.000,E1 124.405} C_DIS
LIN {X -0.081,Y -323.531,Z 1392.688,A 0.000,B 0.000,C 90.000,E1 123.913} C_DIS
LIN {X -0.001,Y -325.048,Z 1392.687,A 0.000,B 0.000,C 90.000,E1 123.579} C_DIS
LIN {X 0.081,Y -339.185,Z 1392.666,A 0.000,B 0.000,C 90.000,E1 119.795} C_DIS
LIN {X -0.059,Y -351.288,Z 1392.650,A 0.000,B 0.000,C 90.000,E1 117.052} C_DIS
LIN {X -0.010,Y -364.856,Z 1392.635,A 0.000,B 0.000,C 90.000,E1 114.335} C_DIS
LIN {X 0.030,Y -378.246,Z 1392.622,A 0.000,B 0.000,C 90.000,E1 111.972} C_DIS
LIN {X -0.100,Y -392.982,Z 1392.609,A 0.000,B 0.000,C 90.000,E1 109.685} C_DIS
LIN {X 0.110,Y -409.165,Z 1392.597,A 0.000,B 0.000,C 90.000,E1 107.402} C_DIS
LIN {X -0.183,Y -426.912,Z 1392.585,A 0.000,B 0.000,C 90.000,E1 105.245} C_DIS
LIN {X 0.216,Y -446.256,Z 1392.573,A 0.000,B 0.000,C 90.000,E1 103.063} C_DIS
LIN {X -0.144,Y -466.426,Z 1392.562,A 0.000,B 0.000,C 90.000,E1 101.130} C_DIS
LIN {X 0.099,Y -484.333,Z 1392.553,A 0.000,B 0.000,C 90.000,E1 99.500} C_DIS
LIN {X 0.131,Y -486.246,Z 1392.552,A 0.000,B 0.000,C 90.000,E1 99.265} C_DIS
LIN {X 0.160,Y -487.703,Z 1392.550,A 0.000,B 0.000,C 90.000,E1 99.029} C_DIS
LIN {X -0.126,Y -489.729,Z 1392.547,A 0.000,B 0.000,C 90.000,E1 98.568} C_DIS
LIN {X 0.081,Y -490.604,Z 1392.545,A 0.000,B 0.000,C 90.000,E1 98.049} C_DIS
LIN {X -0.184,Y -490.481,Z 1392.542,A 0.000,B 0.000,C 90.000,E1 97.587} C_DIS
LIN {X 0.044,Y -489.344,Z 1392.539,A 0.000,B 0.000,C 90.000,E1 97.068} C_DIS
LIN {X -0.056,Y -488.343,Z 1392.538,A 0.000,B 0.000,C 90.000,E1 96.834} C_DIS
LIN {X -0.214,Y -486.987,Z 1392.537,A 0.000,B 0.000,C 90.000,E1 96.606} C_DIS
LIN {X -0.221,Y -467.254,Z 1392.520,A 0.000,B 0.000,C 90.000,E1 93.612} C_DIS
LIN {X -0.057,Y -457.257,Z 1392.511,A 0.000,B 0.000,C 90.000,E1 92.064} C_DIS
LIN {X 0.181,Y -437.969,Z 1392.494,A 0.000,B 0.000,C 90.000,E1 88.912} C_DIS
LIN {X 0.136,Y -425.926,Z 1392.482,A 0.000,B 0.000,C 90.000,E1 86.788} C_DIS
LIN {X 0.046,Y -416.810,Z 1392.473,A 0.000,B 0.000,C 90.000,E1 85.179} C_DIS
LIN {X -0.044,Y -404.458,Z 1392.461,A 0.000,B 0.000,C 90.000,E1 82.996} C_DIS
LIN {X -0.028,Y -395.068,Z 1392.452,A 0.000,B 0.000,C 90.000,E1 81.319} C_DIS
LIN {X -0.115,Y -385.511,Z 1392.442,A 0.000,B 0.000,C 90.000,E1 79.634} C_DIS
LIN {X 0.095,Y -372.553,Z 1392.430,A 0.000,B 0.000,C 90.000,E1 77.297} C_DIS
LIN {X 0.209,Y -362.786,Z 1392.420,A 0.000,B 0.000,C 90.000,E1 75.519} C_DIS
LIN {X 0.149,Y -352.833,Z 1392.410,A 0.000,B 0.000,C 90.000,E1 73.740} C_DIS
LIN {X 0.008,Y -342.848,Z 1392.400,A 0.000,B 0.000,C 90.000,E1 71.945} C_DIS
LIN {X 0.201,Y -331.129,Z 1392.388,A 0.000,B 0.000,C 90.000,E1 69.752} C_DIS
LIN {X 0.081,Y -314.953,Z 1392.370,A 0.000,B 0.000,C 90.000,E1 66.613} C_DIS
LIN {X -0.017,Y -300.214,Z 1392.352,A 0.000,B 0.000,C 90.000,E1 63.384} C_DIS
LIN {X 0.001,Y -287.289,Z 1392.334,A 0.000,B 0.000,C 90.000,E1 60.049} C_DIS
LIN {X 0.010,Y -274.823,Z 1392.313,A 0.000,B 0.000,C 90.000,E1 56.294} C_DIS
LIN {X 0.097,Y -266.486,Z 1392.297,A 0.000,B 0.000,C 90.000,E1 53.497} C_DIS
LIN {X -0.030,Y -256.636,Z 1392.278,A 0.000,B 0.000,C 90.000,E1 49.989} C_DIS
LIN {X -0.004,Y -249.166,Z 1392.262,A 0.000,B 0.000,C 90.000,E1 47.106} C_DIS
LIN {X -0.047,Y -240.581,Z 1392.241,A 0.000,B 0.000,C 90.000,E1 43.461} C_DIS
LIN {X 0.026,Y -232.771,Z 1392.221,A 0.000,B 0.000,C 90.000,E1 39.725} C_DIS
LIN {X -0.038,Y -225.906,Z 1392.200,A 0.000,B 0.000,C 90.000,E1 35.964} C_DIS
LIN {X -0.031,Y -219.914,Z 1392.178,A 0.000,B 0.000,C 90.000,E1 32.133} C_DIS
LIN {X 0.066,Y -214.848,Z 1392.157,A 0.000,B 0.000,C 90.000,E1 28.231} C_DIS
LIN {X 0.109,Y -210.015,Z 1392.131,A 0.000,B 0.000,C 90.000,E1 23.515} C_DIS
LIN {X -0.004,Y -206.077,Z 1392.100,A 0.000,B 0.000,C 90.000,E1 18.000} C_DIS
LIN {X 0.010,Y -203.985,Z 1392.078,A 0.000,B 0.000,C 90.000,E1 14.008} C_DIS
LIN {X -0.106,Y -202.511,Z 1392.060,A 0.000,B 0.000,C 90.000,E1 10.838} C_DIS
LIN {X 0.046,Y -200.893,Z 1392.038,A 0.000,B 0.000,C 90.000,E1 6.777} C_DIS
LIN {X 0.025,Y -199.622,Z 1392.015,A 0.000,B 0.000,C 90.000,E1 2.751} C_DIS
LIN {X -0.062,Y -198.607,Z 1391.993,A 0.000,B 0.000,C 90.000,E1 358.740} C_DIS
LIN {X -0.015,Y -197.922,Z 1391.961,A 0.000,B 0.000,C 90.000,E1 353.053} C_DIS
LIN {X -0.099,Y -198.700,Z 1391.925,A 0.000,B 0.000,C 90.000,E1 346.589} C_DIS
LIN {X 0.110,Y -201.527,Z 1391.889,A 0.000,B 0.000,C 90.000,E1 340.061} C_DIS
LIN {X -0.029,Y -205.383,Z 1391.863,A 0.000,B 0.000,C 90.000,E1 335.281} C_DIS
LIN {X -0.063,Y -209.813,Z 1391.840,A 0.000,B 0.000,C 90.000,E1 331.307} C_DIS
LIN {X 0.076,Y -215.425,Z 1391.819,A 0.000,B 0.000,C 90.000,E1 327.327} C_DIS
LIN {X 0.122,Y -220.883,Z 1391.801,A 0.000,B 0.000,C 90.000,E1 324.196} C_DIS
LIN {X -0.101,Y -227.237,Z 1391.784,A 0.000,B 0.000,C 90.000,E1 321.170} C_DIS
LIN {X 0.091,Y -234.521,Z 1391.767,A 0.000,B 0.000,C 90.000,E1 318.081} C_DIS
LIN {X -0.069,Y -243.670,Z 1391.749,A 0.000,B 0.000,C 90.000,E1 314.757} C_DIS
LIN {X 0.037,Y -251.583,Z 1391.734,A 0.000,B 0.000,C 90.000,E1 312.162} C_DIS
LIN {X 0.031,Y -261.747,Z 1391.718,A 0.000,B 0.000,C 90.000,E1 309.277} C_DIS
LIN {X 0.081,Y -274.583,Z 1391.701,A 0.000,B 0.000,C 90.000,E1 306.091} C_DIS
LIN {X -0.147,Y -282.455,Z 1391.691,A 0.000,B 0.000,C 90.000,E1 304.405} C_DIS
LIN {X -0.015,Y -291.247,Z 1391.682,A 0.000,B 0.000,C 90.000,E1 302.673} C_DIS
LIN {X -0.059,Y -299.158,Z 1391.674,A 0.000,B 0.000,C 90.000,E1 301.337} C_DIS
LIN {X 0.027,Y -310.159,Z 1391.665,A 0.000,B 0.000,C 90.000,E1 299.667} C_DIS
LIN {X 0.082,Y -320.092,Z 1391.658,A 0.000,B 0.000,C 90.000,E1 298.359} C_DIS
LIN {X -0.013,Y -336.044,Z 1391.647,A 0.000,B 0.000,C 90.000,E1 296.539} C_DIS
LIN {X -0.034,Y -349.559,Z 1391.639,A 0.000,B 0.000,C 90.000,E1 295.079} C_DIS
LIN {X -0.019,Y -362.855,Z 1391.631,A 0.000,B 0.000,C 90.000,E1 293.643} C_DIS
LIN {X -0.116,Y -373.366,Z 1391.625,A 0.000,B 0.000,C 90.000,E1 292.514} C_DIS
LIN {X -0.049,Y -383.609,Z 1391.619,A 0.000,B 0.000,C 90.000,E1 291.354} C_DIS
LIN {X -0.069,Y -395.971,Z 1391.611,A 0.000,B 0.000,C 90.000,E1 289.939} C_DIS
LIN {X 0.115,Y -415.848,Z 1391.598,A 0.000,B 0.000,C 90.000,E1 287.692} C_DIS
LIN {X 0.207,Y -423.176,Z 1391.594,A 0.000,B 0.000,C 90.000,E1 286.858} C_DIS
LIN {X -0.044,Y -429.937,Z 1391.589,A 0.000,B 0.000,C 90.000,E1 286.079} C_DIS
LIN {X 0.171,Y -435.949,Z 1391.585,A 0.000,B 0.000,C 90.000,E1 285.245} C_DIS
LIN {X -0.087,Y -441.174,Z 1391.580,A 0.000,B 0.000,C 90.000,E1 284.481} C_DIS
LIN {X 0.017,Y -444.187,Z 1391.577,A 0.000,B 0.000,C 90.000,E1 283.939} C_DIS
LIN {X -0.176,Y -447.949,Z 1391.573,A 0.000,B 0.000,C 90.000,E1 283.175} C_DIS
LIN {X -0.138,Y -450.060,Z 1391.570,A 0.000,B 0.000,C 90.000,E1 282.647} C_DIS
LIN {X -0.086,Y -451.846,Z 1391.567,A 0.000,B 0.000,C 90.000,E1 282.119} C_DIS
LIN {X -0.028,Y -453.235,Z 1391.564,A 0.000,B 0.000,C 90.000,E1 281.591} C_DIS
LIN {X -0.048,Y -454.259,Z 1391.562,A 0.000,B 0.000,C 90.000,E1 281.074} C_DIS
LIN {X 0.029,Y -454.911,Z 1391.559,A 0.000,B 0.000,C 90.000,E1 280.546} C_DIS
LIN {X 0.111,Y -455.152,Z 1391.556,A 0.000,B 0.000,C 90.000,E1 280.018} C_DIS
LIN {X 0.117,Y -454.908,Z 1391.553,A 0.000,B 0.000,C 90.000,E1 279.500} C_DIS
LIN {X 0.199,Y -454.257,Z 1391.550,A 0.000,B 0.000,C 90.000,E1 278.973} C_DIS
LIN {X 0.209,Y -453.078,Z 1391.547,A 0.000,B 0.000,C 90.000,E1 278.454} C_DIS
LIN {X -0.230,Y -451.345,Z 1391.544,A 0.000,B 0.000,C 90.000,E1 277.992} C_DIS
LIN {X 0.025,Y -450.284,Z 1391.543,A 0.000,B 0.000,C 90.000,E1 277.701} C_DIS
LIN {X 0.020,Y -447.575,Z 1391.540,A 0.000,B 0.000,C 90.000,E1 277.182} C_DIS
LIN {X -0.002,Y -444.102,Z 1391.537,A 0.000,B 0.000,C 90.000,E1 276.663} C_DIS
LIN {X 0.229,Y -442.063,Z 1391.536,A 0.000,B 0.000,C 90.000,E1 276.372} C_DIS
LIN {X 0.178,Y -437.129,Z 1391.533,A 0.000,B 0.000,C 90.000,E1 275.853} C_DIS
LIN {X 0.229,Y -431.103,Z 1391.530,A 0.000,B 0.000,C 90.000,E1 275.334} C_DIS
LIN {X -0.093,Y -424.914,Z 1391.527,A 0.000,B 0.000,C 90.000,E1 274.935} C_DIS
LIN {X -0.001,Y -418.357,Z 1391.525,A 0.000,B 0.000,C 90.000,E1 274.531} C_DIS
LIN {X 0.036,Y -411.778,Z 1391.523,A 0.000,B 0.000,C 90.000,E1 274.188} C_DIS
LIN {X 0.192,Y -401.854,Z 1391.521,A 0.000,B 0.000,C 90.000,E1 273.726} C_DIS
LIN {X -0.099,Y -392.011,Z 1391.519,A 0.000,B 0.000,C 90.000,E1 273.383} C_DIS
LIN {X 0.018,Y -378.836,Z 1391.516,A 0.000,B 0.000,C 90.000,E1 272.922} C_DIS
LIN {X -0.173,Y -371.633,Z 1391.515,A 0.000,B 0.000,C 90.000,E1 272.751} C_DIS
LIN {X 0.134,Y -360.629,Z 1391.514,A 0.000,B 0.000,C 90.000,E1 272.465} C_DIS
LIN {X 0.022,Y -353.039,Z 1391.513,A 0.000,B 0.000,C 90.000,E1 272.350} C_DIS
LIN {X 0.026,Y -343.441,Z 1391.512,A 0.000,B 0.000,C 90.000,E1 272.236} C_DIS
LIN {X 0.057,Y -328.251,Z 1391.512,A 0.000,B 0.000,C 90.000,E1 272.121} C_DIS
LIN {X -0.055,Y -322.433,Z 1391.512,A 0.000,B 0.000,C 90.000,E1 272.121} C_DIS
LIN {X -0.055,Y -181.245,Z 1391.512,A 0.000,B 0.000,C 90.000,E1 272.121} C_DIS
LIN {X 0.069,Y -181.579,Z 1391.502,A 0.000,B 0.000,C 90.000,E1 270.344} C_DIS
LIN {X 0.045,Y -180.904,Z 1391.474,A 0.000,B 0.000,C 90.000,E1 265.298} C_DIS
LIN {X -0.006,Y -180.250,Z 1391.465,A 0.000,B 0.000,C 90.000,E1 263.628} C_DIS
LIN {X 0.013,Y -178.740,Z 1391.441,A 0.000,B 0.000,C 90.000,E1 259.398} C_DIS
LIN {X -0.089,Y -175.787,Z 1391.413,A 0.000,B 0.000,C 90.000,E1 254.338} C_DIS
LIN {X -0.094,Y -171.972,Z 1391.384,A 0.000,B 0.000,C 90.000,E1 249.209} C_DIS
LIN {X -0.055,Y -171.372,Z 1391.380,A 0.000,B 0.000,C 90.000,E1 248.337} C_DIS
LIN {X -0.069,Y -167.618,Z 1391.356,A 0.000,B 0.000,C 90.000,E1 244.024} C_DIS
LIN {X -0.054,Y -166.269,Z 1391.346,A 0.000,B 0.000,C 90.000,E1 242.281} C_DIS
LIN {X -0.059,Y -163.021,Z 1391.327,A 0.000,B 0.000,C 90.000,E1 238.791} C_DIS
